# B&R Automation Studio project NAEUL004C00R13L518F00 (part 44)

#### Act_Main.st - Do Not Change!!!
```iecst
(** 2019-10-30 **)
ACTION Act_Main:

	fbInit.bOnDirMod	:= tylocalMagConv2Clp.In.bOnDirMod;
	fbInit.tMtrOffDlyTm	:= tylocalMagConv2Clp.In.tMtrOffDlyTm;
	fbEnt.bOnDirMod		:= tylocalMagConv2Clp.In.bOnDirMod;
	fbEnt.tMtrOffDlyTm	:= tylocalMagConv2Clp.In.tMtrOffDlyTm;
	fbPreExit.bOnDirMod		:= tylocalMagConv2Clp.In.bOnDirMod;
	fbPreExit.tMtrOffDlyTm	:= tylocalMagConv2Clp.In.tMtrOffDlyTm;
	fbExit.bOnDirMod	:= tylocalMagConv2Clp.In.bOnDirMod;
	fbExit.tMtrOffDlyTm	:= tylocalMagConv2Clp.In.tMtrOffDlyTm;
	fbExit1.bOnDirMod		:= tylocalMagConv2Clp.In.bOnDirMod;
	fbExit1.tMtrOffDlyTm	:= tylocalMagConv2Clp.In.tMtrOffDlyTm;
	fbFixClprClampChk.tTimeOut	:= tylocalMagConv2Clp.In.tClprClampTO;
	fbFixClprUnclampChk.tTimeOut	:= tylocalMagConv2Clp.In.tClprUnclampTO;
	fbRmtClprClampChk.tTimeOut	:= tylocalMagConv2Clp.In.tClprClampTO;
	fbRmtClprUnclampChk.tTimeOut	:= tylocalMagConv2Clp.In.tClprUnclampTO;
	fbClprDlyTm.PT	:= tylocalMagConv2Clp.In.tMtrOffDlyTm / 2;
	//Set tylocalMagConv2Clp.In.eAct
	IF tylocalMagConv2Clp.Out.eStatus = Idle OR tylocalMagConv2Clp.Out.eStatus = Busy OR tylocalMagConv2Clp.Out.eStatus = Done THEN
		tylocalMagConv2Clp.Out.eStat	:= tylocalMagConv2Clp.In.eAct;
	END_IF

	IF eStatOld <> tylocalMagConv2Clp.Out.eStat THEN
		fbInit(bEn := FALSE);
		fbEnt(bEn := FALSE);
		fbPreExit(bEn := FALSE);
		fbExit(bEn := FALSE);
		fbExit1(bEn := FALSE);
		fbStop(bEn := FALSE);
		fbFixClprClampChk(bEn := FALSE);
		fbFixClprUnclampChk(bEn := FALSE);
		fbRmtClprClampChk(bEn := FALSE);
		fbRmtClprUnclampChk(bEn := FALSE);
		fbClprDlyTm(IN := FALSE);
		fbFixClprDly(IN := FALSE);
		fbWidthChk(IN := FALSE);
		fbClampTim(IN := FALSE);

		IF eStatOld <> MagConv2ClpActIdle
			AND eStatOld <> MagConv2ClpActSetMtrSigOnOrLToR
			AND eStatOld <> MagConv2ClpActSetMtrDirOrRToL
			AND eStatOld <> MagConv2ClpActRstMtrSigOnOrLToR
			AND eStatOld <> MagConv2ClpActRstMtrDirOrRToL
			AND eStatOld <> MagConv2ClpActSetMtrAll
			AND eStatOld <> MagConv2ClpActRstMtrAll THEN

			tylocalMagConv2Clp.Out.bMtrSigOnOrLToR	:= FALSE;
			tylocalMagConv2Clp.Out.bMtrDirOrRToL	:= FALSE;

		END_IF

		usiStep		:= 0;
		usiSubStep	:= 0;
		usiPrevStep := 0;
		bReachEnd	:= FALSE;

		tylocalMagConv2Clp.Out.sStatTxt	:= a_sStatText[tylocalMagConv2Clp.Out.eStat];

		eStatOld	:= tylocalMagConv2Clp.Out.eStat;

		tylocalMagConv2Clp.Out.eStatus		:= Busy;
	END_IF

	//Main
	CASE tylocalMagConv2Clp.Out.eStat OF

		MagConv2ClpActIdle:
			IF EDGENEG(tylocalMagConv2Clp.In.bManual) THEN
				tylocalMagConv2Clp.Out.bMtrSigOnOrLToR	:= FALSE;
				tylocalMagConv2Clp.Out.bMtrDirOrRToL	:= FALSE;
			END_IF

			tylocalMagConv2Clp.Out.eStatus	:= Idle;

		MagConv2ClpActInit:
			IF tylocalMagConv2Clp.Out.eStatus = Idle OR tylocalMagConv2Clp.Out.eStatus = Busy THEN

				tylocalMagConv2Clp.Out.eStatus	:= Busy;

				//Magazine Conveyor Init Run
				//Detect Have Magazine
				IF tylocalMagConv2Clp.In.bLeftSen OR tylocalMagConv2Clp.In.bRightSen THEN
					tylocalMagConv2Clp.Out.bHvMag	:= TRUE;
				ELSE
					tylocalMagConv2Clp.Out.bHvMag	:= FALSE;
				END_IF

				fbInit.bConvLToR	:= (tylocalMagConv2Clp.In.eDirection = ConvDirLToR) OR (tylocalMagConv2Clp.In.eDirection = ConvDirLToL);
				fbInit.tTxDlyTm		:= DINT_TO_TIME(tylocalMagConv2Clp.In.diInitTm);

				IF fbInit.bConvLToR = TRUE THEN
					fbInit.bEndSen	:= tylocalMagConv2Clp.In.bRightSen;
				ELSE
					fbInit.bEndSen	:= tylocalMagConv2Clp.In.bLeftSen;
				END_IF

				fbInit(bEn := TRUE);

				tylocalMagConv2Clp.Out.bMtrSigOnOrLToR	:= fbInit.bMtrSigOnOrLToR;
				tylocalMagConv2Clp.Out.bMtrDirOrRToL	:= fbInit.bMtrDirOrRToL;

				IF fbInit.udiStatus = 0 THEN
					IF fbInit.bConvLToR = TRUE THEN
						IF tylocalMagConv2Clp.Out.bHvMag = TRUE AND tylocalMagConv2Clp.In.bRightSen = FALSE THEN
							udiStatus	:= 10000;	//Magazine Detected But Not Present At Outlet Sensor (L - R) While Magazine Conveyor Initial
							tylocalMagConv2Clp.Out.eStatus		:= Error;
						ELSE
							tylocalMagConv2Clp.Out.eStatus	:= Done;
						END_IF
					ELSE
						IF tylocalMagConv2Clp.Out.bHvMag = TRUE AND tylocalMagConv2Clp.In.bLeftSen = FALSE THEN
							udiStatus	:= 10001;	//Magazine Detected But Not Present At Outlet Sensor (R - L) While Magazine Conveyor Initial
							tylocalMagConv2Clp.Out.eStatus		:= Error;
						ELSE
							tylocalMagConv2Clp.Out.eStatus	:= Done;
						END_IF
					END_IF
				ELSIF fbInit.udiStatus < 65534 THEN
					udiStatus	:= fbInit.udiStatus;
					tylocalMagConv2Clp.Out.eStatus		:= Error;
				END_IF
			END_IF

		MagConv2ClpActInitStopClp:
			IF tylocalMagConv2Clp.Out.eStatus = Idle OR tylocalMagConv2Clp.Out.eStatus = Busy THEN

				tylocalMagConv2Clp.Out.eStatus	:= Busy;

				CASE usiStep OF
					0:	//Unclamp
						tylocalMagConv2Clp.Out.bFixClprClampCtrl	:= FALSE;
						tylocalMagConv2Clp.Out.bRmtClprClampCtrl	:= FALSE;
						tylocalMagConv2Clp.Out.bFixClprUnClampCtrl	:= TRUE;
						tylocalMagConv2Clp.Out.bRmtClprUnClampCtrl	:= TRUE;

						fbFixClprUnclampChk.bExtSen		:= tylocalMagConv2Clp.In.bFixClprClampSen;
						fbFixClprUnclampChk.bRetSen		:= tylocalMagConv2Clp.In.bFixClprUnclampSen;
						fbFixClprUnclampChk.bRetSafety	:= tylocalMagConv2Clp.In.bFixClprUnclampSafetySen;
						fbFixClprUnclampChk(bEn := TRUE);

						fbRmtClprUnclampChk.bExtSen		:= tylocalMagConv2Clp.In.bRmtClprClampSen;
						fbRmtClprUnclampChk.bRetSen		:= tylocalMagConv2Clp.In.bRmtClprUnclampSen;
						fbRmtClprUnclampChk.bRetSafety	:= tylocalMagConv2Clp.In.bRmtClprUnclampSafetySen;
						fbRmtClprUnclampChk(bEn := TRUE);

						IF fbFixClprUnclampChk.udiStatus = 0 AND fbRmtClprUnclampChk.udiStatus = 0 THEN
							usiStep	:= 1;
						ELSIF (fbFixClprUnclampChk.udiStatus > 0 AND fbFixClprUnclampChk.udiStatus < 65534) OR (fbRmtClprUnclampChk.udiStatus > 0 AND fbRmtClprUnclampChk.udiStatus < 65534) THEN
							tylocalMagConv2Clp.Out.bFixClprClampCtrl	:= FALSE;
							tylocalMagConv2Clp.Out.bRmtClprClampCtrl	:= FALSE;
							tylocalMagConv2Clp.Out.bFixClprUnClampCtrl	:= FALSE;
							tylocalMagConv2Clp.Out.bRmtClprUnClampCtrl	:= FALSE;

							tylocalMagConv2Clp.Out.eStatus	:= Error;

							IF fbFixClprUnclampChk.udiStatus = 1504 OR fbRmtClprUnclampChk.udiStatus = 1504 THEN
								udiStatus	:= 10002;	//Clamper Clamp Sensor Off Time Out In Unclamp Check While Conveyor Initial With Clamper
							ELSIF fbFixClprUnclampChk.udiStatus = 1505 OR fbRmtClprUnclampChk.udiStatus = 1505 THEN
								udiStatus	:= 10003;	//Clamper Unclamp Sensor On Time Out In Unclamp Check While Conveyor Initial With Clamper
							ELSIF fbFixClprUnclampChk.udiStatus = 1508 OR fbRmtClprUnclampChk.udiStatus = 1508 THEN
								udiStatus	:= 10004;	//Clamper Unclamp Safety Sensor Error In Unclamp Check While Conveyor Initial With Clamper
							ELSE
								IF fbFixClprUnclampChk.udiStatus > 0 AND fbFixClprUnclampChk.udiStatus < 65534 THEN
									udiStatus	:= fbFixClprUnclampChk.udiStatus;
								ELSIF fbRmtClprUnclampChk.udiStatus > 0 AND fbRmtClprUnclampChk.udiStatus < 65534 THEN
									udiStatus	:= fbRmtClprUnclampChk.udiStatus;
								END_IF
							END_IF
						END_IF

					1:	//Magazine Conveyor Init Run
						//Detect Have Magazine
						IF tylocalMagConv2Clp.In.bLeftSen OR tylocalMagConv2Clp.In.bRightSen THEN
							tylocalMagConv2Clp.Out.bHvMag	:= TRUE;
						ELSE
							tylocalMagConv2Clp.Out.bHvMag	:= FALSE;
						END_IF

						fbInit.bConvLToR	:= (tylocalMagConv2Clp.In.eDirection = ConvDirLToR) OR (tylocalMagConv2Clp.In.eDirection = ConvDirLToL);
						fbInit.tTxDlyTm		:= DINT_TO_TIME(tylocalMagConv2Clp.In.diInitTm);

						IF fbInit.bConvLToR = TRUE THEN
							fbInit.bEndSen	:= tylocalMagConv2Clp.In.bRightSen;
						ELSE
							fbInit.bEndSen	:= tylocalMagConv2Clp.In.bLeftSen;
						END_IF

						fbInit(bEn := TRUE);

						tylocalMagConv2Clp.Out.bMtrSigOnOrLToR	:= fbInit.bMtrSigOnOrLToR;
						tylocalMagConv2Clp.Out.bMtrDirOrRToL	:= fbInit.bMtrDirOrRToL;

						IF fbInit.udiStatus = 0 THEN
							IF fbInit.bConvLToR = TRUE THEN
								IF tylocalMagConv2Clp.Out.bHvMag = TRUE AND tylocalMagConv2Clp.In.bRightSen = FALSE THEN
									udiStatus	:= 10005;	//Magazine Detected But Not Present At Outlet Sensor (L - R) While Conveyor Initial With Clamper
									tylocalMagConv2Clp.Out.eStatus		:= Error;
								ELSE
									usiStep	:= 2;
								END_IF
							ELSE
								IF tylocalMagConv2Clp.Out.bHvMag = TRUE AND tylocalMagConv2Clp.In.bLeftSen = FALSE THEN
									udiStatus	:= 10006;	//Magazine Detected But Not Present At Outlet Sensor (R - L) While Conveyor Initial With Clamper
									tylocalMagConv2Clp.Out.eStatus		:= Error;
								ELSE
									usiStep	:= 2;
								END_IF
							END_IF
						ELSIF fbInit.udiStatus < 65534 THEN
							udiStatus	:= fbInit.udiStatus;
							tylocalMagConv2Clp.Out.eStatus		:= Error;
						END_IF

					2:	//Check If Have Magazine
						IF tylocalMagConv2Clp.Out.bHvMag = TRUE THEN
							fbWidthChk(IN := NOT tylocalMagConv2Clp.In.bWidthChkInterrupt);
							IF tylocalMagConv2Clp.In.bWidthChkInterrupt = FALSE THEN
								IF fbWidthChk.Q THEN
									udiStatus := 10048;
									tylocalMagConv2Clp.Out.eStatus	  := Error; //Safety Sensor Is Deactivated Before Clamp
								END_IF
							ELSIF tylocalMagConv2Clp.In.bWidthChkInterrupt THEN
								usiStep	  := 3;
							END_IF
						ELSE
							tylocalMagConv2Clp.Out.eStatus	:= Done;
						END_IF

					3:	//Fix Clamp
						tylocalMagConv2Clp.Out.bFixClprClampCtrl	:= TRUE;
						tylocalMagConv2Clp.Out.bFixClprUnClampCtrl	:= FALSE;

						fbFixClprClampChk.bExtSen		:= tylocalMagConv2Clp.In.bFixClprClampSen;
						fbFixClprClampChk.bRetSen		:= tylocalMagConv2Clp.In.bFixClprUnclampSen;
						fbFixClprClampChk.bExtSafety	:= tylocalMagConv2Clp.In.bFixClprClampSafetySen;
						fbFixClprClampChk(bEn := TRUE);

						IF fbFixClprClampChk.udiStatus = 0 THEN
							fbFixClprDly (IN := TRUE);
							IF  fbFixClprDly.Q THEN
								fbFixClprDly (IN := FALSE);
								usiStep	:= 4;
							END_IF

						ELSIF fbFixClprClampChk.udiStatus < 65534 THEN
							tylocalMagConv2Clp.Out.bFixClprClampCtrl	:= FALSE;
							tylocalMagConv2Clp.Out.bFixClprUnClampCtrl	:= FALSE;

							tylocalMagConv2Clp.Out.eStatus	:= Error;

							IF fbFixClprClampChk.udiStatus = 1503 THEN
								udiStatus	:= 10007;	//Clamper Clamp Sensor On Time Out In Clamp Check While Conveyor Initial With Clamper
							ELSIF fbFixClprClampChk.udiStatus = 1506 THEN
								udiStatus	:= 10008;	//Clamper Unclamp Sensor Off Time Out In Clamp Check While Conveyor Initial With Clamper
							ELSIF fbFixClprClampChk.udiStatus = 1507 THEN
								udiStatus	:= 10009;	//Clamper Clamp Safety Sensor Error In Clamp Check While Conveyor Initial With Clamper
							ELSE
								udiStatus	:= fbFixClprClampChk.udiStatus;
							END_IF
						END_IF

					4:	//Remote Clamp
						tylocalMagConv2Clp.Out.bRmtClprClampCtrl	:= TRUE;
						tylocalMagConv2Clp.Out.bRmtClprUnClampCtrl	:= FALSE;

						fbRmtClprClampChk.bExtSen		:= tylocalMagConv2Clp.In.bRmtClprClampSen;
						fbRmtClprClampChk.bRetSen		:= tylocalMagConv2Clp.In.bRmtClprUnclampSen;
						fbRmtClprClampChk.bExtSafety	:= tylocalMagConv2Clp.In.bRmtClprClampSafetySen;
						fbRmtClprClampChk(bEn := TRUE);

						IF fbRmtClprClampChk.udiStatus = 0 THEN
							tylocalMagConv2Clp.Out.eStatus	:= Done;

						ELSIF fbRmtClprClampChk.udiStatus < 65534 THEN
							tylocalMagConv2Clp.Out.bRmtClprClampCtrl	:= FALSE;
							tylocalMagConv2Clp.Out.bRmtClprUnClampCtrl	:= FALSE;
							tylocalMagConv2Clp.Out.eStatus	:= Error;

							IF fbRmtClprClampChk.udiStatus = 1503 THEN
								udiStatus	:= 10007;	//Clamper Clamp Sensor On Time Out In Clamp Check While Conveyor Initial With Clamper
							ELSIF fbRmtClprClampChk.udiStatus = 1506 THEN
								udiStatus	:= 10008;	//Clamper Unclamp Sensor Off Time Out In Clamp Check While Conveyor Initial With Clamper
							ELSIF fbRmtClprClampChk.udiStatus = 1507 THEN
								udiStatus	:= 10009;	//Clamper Clamp Safety Sensor Error In Clamp Check While Conveyor Initial With Clamper
							ELSE
								udiStatus	:= fbRmtClprClampChk.udiStatus;
							END_IF
						END_IF

				END_CASE
			END_IF

		MagConv2ClpActInitClpStop:
			IF tylocalMagConv2Clp.Out.eStatus = Idle OR tylocalMagConv2Clp.Out.eStatus = Busy THEN

				tylocalMagConv2Clp.Out.eStatus	:= Busy;

				CASE usiStep OF
					0:	//Unclamp
						tylocalMagConv2Clp.Out.bFixClprClampCtrl	:= FALSE;
						tylocalMagConv2Clp.Out.bRmtClprClampCtrl	:= FALSE;
						tylocalMagConv2Clp.Out.bFixClprUnClampCtrl	:= TRUE;
						tylocalMagConv2Clp.Out.bRmtClprUnClampCtrl	:= TRUE;

						fbFixClprUnclampChk.bExtSen		:= tylocalMagConv2Clp.In.bFixClprClampSen;
						fbFixClprUnclampChk.bRetSen		:= tylocalMagConv2Clp.In.bFixClprUnclampSen;
						fbFixClprUnclampChk.bRetSafety	:= tylocalMagConv2Clp.In.bFixClprUnclampSafetySen;
						fbFixClprUnclampChk(bEn := TRUE);

						fbRmtClprUnclampChk.bExtSen		:= tylocalMagConv2Clp.In.bRmtClprClampSen;
						fbRmtClprUnclampChk.bRetSen		:= tylocalMagConv2Clp.In.bRmtClprUnclampSen;
						fbRmtClprUnclampChk.bRetSafety	:= tylocalMagConv2Clp.In.bRmtClprUnclampSafetySen;
						fbRmtClprUnclampChk(bEn := TRUE);

						IF fbFixClprUnclampChk.udiStatus = 0 AND fbRmtClprUnclampChk.udiStatus = 0 THEN
							usiStep	:= 1;
						ELSIF (fbFixClprUnclampChk.udiStatus > 0 AND fbFixClprUnclampChk.udiStatus < 65534) OR (fbRmtClprUnclampChk.udiStatus > 0 AND fbRmtClprUnclampChk.udiStatus < 65534) THEN
							tylocalMagConv2Clp.Out.bFixClprClampCtrl	:= FALSE;
							tylocalMagConv2Clp.Out.bRmtClprClampCtrl	:= FALSE;
							tylocalMagConv2Clp.Out.bFixClprUnClampCtrl	:= FALSE;
							tylocalMagConv2Clp.Out.bRmtClprUnClampCtrl	:= FALSE;

							tylocalMagConv2Clp.Out.eStatus	:= Error;

							IF fbFixClprUnclampChk.udiStatus = 1504 OR fbRmtClprUnclampChk.udiStatus = 1504 THEN
								udiStatus	:= 10002;	//Clamper Clamp Sensor Off Time Out In Unclamp Check While Conveyor Initial With Clamper
							ELSIF fbFixClprUnclampChk.udiStatus = 1505 OR fbRmtClprUnclampChk.udiStatus = 1505 THEN
								udiStatus	:= 10003;	//Clamper Unclamp Sensor On Time Out In Unclamp Check While Conveyor Initial With Clamper
							ELSIF fbFixClprUnclampChk.udiStatus = 1508 OR fbRmtClprUnclampChk.udiStatus = 1508 THEN
								udiStatus	:= 10004;	//Clamper Unclamp Safety Sensor Error In Unclamp Check While Conveyor Initial With Clamper
							ELSE
								IF fbFixClprUnclampChk.udiStatus > 0 AND fbFixClprUnclampChk.udiStatus < 65534 THEN
									udiStatus	:= fbFixClprUnclampChk.udiStatus;
								ELSIF fbRmtClprUnclampChk.udiStatus > 0 AND fbRmtClprUnclampChk.udiStatus < 65534 THEN
									udiStatus	:= fbRmtClprUnclampChk.udiStatus;
								END_IF
							END_IF
						END_IF

					1:	//Magazine Conveyor Init Run & Clamp
						//Detect Have Magazine
						IF tylocalMagConv2Clp.In.bLeftSen OR tylocalMagConv2Clp.In.bRightSen THEN
							tylocalMagConv2Clp.Out.bHvMag	:= TRUE;
						ELSE
							tylocalMagConv2Clp.Out.bHvMag	:= FALSE;
						END_IF

						fbInit.bConvLToR	:= (tylocalMagConv2Clp.In.eDirection = ConvDirLToR) OR (tylocalMagConv2Clp.In.eDirection = ConvDirLToL);
						fbInit.tTxDlyTm		:= DINT_TO_TIME(tylocalMagConv2Clp.In.diInitTm);

						IF fbInit.bConvLToR = TRUE THEN
							fbInit.bEndSen	:= tylocalMagConv2Clp.In.bRightSen;
						ELSE
							fbInit.bEndSen	:= tylocalMagConv2Clp.In.bLeftSen;
						END_IF

						fbInit(bEn := TRUE);

						tylocalMagConv2Clp.Out.bMtrSigOnOrLToR	:= fbInit.bMtrSigOnOrLToR;
						tylocalMagConv2Clp.Out.bMtrDirOrRToL	:= fbInit.bMtrDirOrRToL;

						IF fbInit.bEndSen = TRUE THEN
							bReachEnd	:= TRUE;
						END_IF

						IF bReachEnd = TRUE THEN
							fbClprDlyTm(IN := TRUE);
							IF fbClprDlyTm.Q = TRUE THEN
								CASE usiSubStep OF
									//	0:	//Fix Clamp
									//										tylocalMagConv2Clp.Out.bFixClprClampCtrl	:= TRUE;

									//										fbFixClprClampChk.bExtSen		:= tylocalMagConv2Clp.In.bFixClprClampSen;
									//										fbFixClprClampChk.bRetSen		:= tylocalMagConv2Clp.In.bFixClprUnclampSen;
									//										fbFixClprClampChk.bExtSafety	:= tylocalMagConv2Clp.In.bFixClprClampSafetySen;
									//										fbFixClprClampChk(bEn := TRUE);
									//
									//										IF fbFixClprClampChk.udiStatus = 0 THEN
									//											usiSubStep	:= 1;
									//										END_IF

									0:	//Remote Clamp
										tylocalMagConv2Clp.Out.bRmtClprClampCtrl	:= TRUE;
										tylocalMagConv2Clp.Out.bRmtClprUnClampCtrl	:= FALSE;
										fbRmtClprClampChk.bExtSen		:= tylocalMagConv2Clp.In.bRmtClprClampSen;
										fbRmtClprClampChk.bRetSen		:= tylocalMagConv2Clp.In.bRmtClprUnclampSen;
										fbRmtClprClampChk.bExtSafety	:= tylocalMagConv2Clp.In.bRmtClprClampSafetySen;
										fbRmtClprClampChk(bEn := TRUE);

										IF fbRmtClprClampChk.udiStatus = 0 THEN
											usiSubStep	:= 1;
										END_IF

									1:

										tylocalMagConv2Clp.Out.bFixClprClampCtrl	:= TRUE;
										tylocalMagConv2Clp.Out.bFixClprUnClampCtrl	:= FALSE;

										fbFixClprClampChk.bExtSen		:= tylocalMagConv2Clp.In.bFixClprClampSen;
										fbFixClprClampChk.bRetSen		:= tylocalMagConv2Clp.In.bFixClprUnclampSen;
										fbFixClprClampChk.bExtSafety	:= tylocalMagConv2Clp.In.bFixClprClampSafetySen;
										fbFixClprClampChk(bEn := TRUE);

								END_CASE
							END_IF
						END_IF

						IF (fbInit.udiStatus = 0) AND ((fbFixClprClampChk.udiStatus = 0 AND fbRmtClprClampChk.udiStatus = 0) OR (bReachEnd = FALSE)) THEN
							IF fbInit.bConvLToR = TRUE THEN
								IF tylocalMagConv2Clp.Out.bHvMag = TRUE AND tylocalMagConv2Clp.In.bRightSen = FALSE THEN
									udiStatus	:= 10041;	//Magazine Detected But Not Present At Outlet Sensor (L - R) While Conveyor Initial With Clamper
									tylocalMagConv2Clp.Out.eStatus		:= Error;
								ELSE
									tylocalMagConv2Clp.Out.eStatus		:= Done;
								END_IF
							ELSE
								IF tylocalMagConv2Clp.Out.bHvMag = TRUE AND tylocalMagConv2Clp.In.bLeftSen = FALSE THEN
									udiStatus	:= 10042;	//Magazine Detected But Not Present At Outlet Sensor (R - L) While Conveyor Initial With Clamper
									tylocalMagConv2Clp.Out.eStatus		:= Error;
								ELSE
									tylocalMagConv2Clp.Out.eStatus		:= Done;
								END_IF
							END_IF

						ELSIF fbInit.udiStatus > 0 AND fbInit.udiStatus < 65534 THEN
							udiStatus	:= fbInit.udiStatus;
							tylocalMagConv2Clp.Out.eStatus		:= Error;

						ELSIF (fbFixClprClampChk.udiStatus > 0 AND fbFixClprClampChk.udiStatus < 65534) OR (fbRmtClprClampChk.udiStatus > 0 AND fbRmtClprClampChk.udiStatus < 65534) THEN
							tylocalMagConv2Clp.Out.bFixClprClampCtrl	:= FALSE;
							tylocalMagConv2Clp.Out.bRmtClprClampCtrl	:= FALSE;
							tylocalMagConv2Clp.Out.bFixClprUnClampCtrl	:= FALSE;
							tylocalMagConv2Clp.Out.bRmtClprUnClampCtrl	:= FALSE;

							tylocalMagConv2Clp.Out.eStatus	:= Error;

							IF fbFixClprClampChk.udiStatus = 1503 OR fbRmtClprClampChk.udiStatus = 1503 THEN
								udiStatus	:= 10043;	//Clamper Clamp Sensor On Time Out In Clamp Check While Conveyor Initial With Clamper
							ELSIF fbFixClprClampChk.udiStatus = 1506 OR fbRmtClprClampChk.udiStatus = 1506 THEN
								udiStatus	:= 10044;	//Clamper Unclamp Sensor Off Time Out In Clamp Check While Conveyor Initial With Clamper
							ELSIF fbFixClprClampChk.udiStatus = 1507 OR fbRmtClprClampChk.udiStatus = 1507 THEN
								udiStatus	:= 10045;	//Clamper Clamp Safety Sensor Error In Clamp Check While Conveyor Initial With Clamper
							ELSE
								IF fbFixClprClampChk.udiStatus > 0 AND fbFixClprClampChk.udiStatus < 65534 THEN
									udiStatus	:= fbFixClprClampChk.udiStatus;
								ELSIF fbRmtClprClampChk.udiStatus > 0 AND fbRmtClprClampChk.udiStatus < 65534 THEN
									udiStatus	:= fbRmtClprClampChk.udiStatus;
								END_IF
							END_IF
						END_IF

				END_CASE
			END_IF

		MagConv2ClpActEnt:
			IF tylocalMagConv2Clp.Out.eStatus = Idle OR tylocalMagConv2Clp.Out.eStatus = Busy THEN

				tylocalMagConv2Clp.Out.eStatus	:= Busy;

				//Detect Have Magazine
				IF tylocalMagConv2Clp.In.bLeftSen OR tylocalMagConv2Clp.In.bRightSen THEN
					tylocalMagConv2Clp.Out.bHvMag	:= TRUE;
				END_IF

				//Conveyor Run
				fbEnt.bConvLToR		:= (tylocalMagConv2Clp.In.eDirection = ConvDirLToR) OR (tylocalMagConv2Clp.In.eDirection = ConvDirLToL);
				fbEnt.tTimeOut		:= DINT_TO_TIME(tylocalMagConv2Clp.In.diTxInTimeOut);

				IF fbEnt.bConvLToR = TRUE THEN
					fbEnt.bEndSen	:= tylocalMagConv2Clp.In.bRightSen;
				ELSE
					fbEnt.bEndSen	:= tylocalMagConv2Clp.In.bLeftSen;
				END_IF

				fbEnt(bEn := TRUE);

				tylocalMagConv2Clp.Out.bMtrSigOnOrLToR	:= fbEnt.bMtrSigOnOrLToR;
				tylocalMagConv2Clp.Out.bMtrDirOrRToL	:= fbEnt.bMtrDirOrRToL;

				IF fbEnt.udiStatus = 0 THEN
					tylocalMagConv2Clp.Out.eStatus		:= Done;
				ELSIF fbEnt.udiStatus < 65534 THEN
					tylocalMagConv2Clp.Out.eStatus		:= Error;

					IF fbEnt.udiStatus = 1101 THEN
						udiStatus	:= 10028;	//Transfer In Time Out While Entering Magazine
					ELSE
						udiStatus	:= fbEnt.udiStatus;
					END_IF
				END_IF

			END_IF

		MagConv2ClpActEntStopClp:
			IF tylocalMagConv2Clp.Out.eStatus = Idle OR tylocalMagConv2Clp.Out.eStatus = Busy THEN

				tylocalMagConv2Clp.Out.eStatus	:= Busy;

				CASE usiStep OF
					0:	//Conveyor Enter
						//Detect Have Magazine
						IF tylocalMagConv2Clp.In.bLeftSen OR tylocalMagConv2Clp.In.bRightSen THEN
							tylocalMagConv2Clp.Out.bHvMag	:= TRUE;
						END_IF

						//Conveyor Run
						fbEnt.bConvLToR		:= (tylocalMagConv2Clp.In.eDirection = ConvDirLToR) OR (tylocalMagConv2Clp.In.eDirection = ConvDirLToL);
						fbEnt.tTimeOut		:= DINT_TO_TIME(tylocalMagConv2Clp.In.diTxInTimeOut);

						IF fbEnt.bConvLToR = TRUE THEN
							fbEnt.bEndSen	:= tylocalMagConv2Clp.In.bRightSen;
						ELSE
							fbEnt.bEndSen	:= tylocalMagConv2Clp.In.bLeftSen;
						END_IF

						fbEnt(bEn := TRUE);

						tylocalMagConv2Clp.Out.bMtrSigOnOrLToR	:= fbEnt.bMtrSigOnOrLToR;
						tylocalMagConv2Clp.Out.bMtrDirOrRToL	:= fbEnt.bMtrDirOrRToL;

						IF fbEnt.udiStatus = 0 THEN
							usiStep	:= 2;
							tRemainingTime := tylocalMagConv2Clp.In.tClprClampTO;

						ELSIF fbEnt.udiStatus < 65534 THEN
							tylocalMagConv2Clp.Out.eStatus	:= Error;

							IF fbEnt.udiStatus = 1101 THEN
								udiStatus	:= 10029;	//Transfer In Time Out While Entering Magazine
							ELSE
								udiStatus	:= fbEnt.udiStatus;
							END_IF
						END_IF
					1: //clamp standby step
						fbFixClprClampChk(bEn:= FALSE);
						fbRmtClprClampChk(bEn:= FALSE);
						fbFixClprUnclampChk(bEn:= FALSE);
						fbRmtClprUnclampChk(bEn := FALSE);
						fbInterrupSenDlyOff(IN:= tylocalMagConv2Clp.In.bWidthChkInterrupt);
						IF fbInterrupSenDlyOff.Q THEN
							IF NOT(tylocalMagConv2Clp.In.bLeftSen) AND NOT(tylocalMagConv2Clp.In.bRightSen) THEN
								tylocalMagConv2Clp.Out.eStatus := Error;
								udiStatus	:= 10049; //Magazine is taken away during the clamp
							ELSIF (tylocalMagConv2Clp.In.bLeftSen AND NOT(tylocalMagConv2Clp.In.bRightSen)) THEN
								fbEnt(bEn := FALSE);
								usiStep := 4;
								IF usiPrevStep <> usiStep THEN
									tRemainingTime := tylocalMagConv2Clp.In.tClprClampTO;
								END_IF
							ELSE
								usiStep := usiPrevStep;
								usiPrevStep := 1;
							END_IF
						END_IF

					2:	//Fix Clamp
						tylocalMagConv2Clp.Out.bFixClprClampCtrl	:= TRUE;
						tylocalMagConv2Clp.Out.bFixClprUnClampCtrl	:= FALSE;

						fbFixClprClampChk.bExtSen		:= tylocalMagConv2Clp.In.bFixClprClampSen;
						fbFixClprClampChk.bRetSen		:= tylocalMagConv2Clp.In.bFixClprUnclampSen ;// OR (usiPrevStep = 1 AND tylocalMagConv2Clp.In.bFixClprClampSen = FALSE);
						fbFixClprClampChk.bExtSafety	:= tylocalMagConv2Clp.In.bFixClprClampSafetySen;
						fbFixClprClampChk(bEn := TRUE);
						IF (tRemainingTime) > T#5s THEN
							fbClampTim(IN:= TRUE,PT:= tRemainingTime );
						ELSE
							fbClampTim(IN:= TRUE,PT:= T#6s);
						END_IF
						IF fbFixClprClampChk.udiStatus = 0 THEN
							fbFixClprDly(IN := TRUE);
							IF  fbFixClprDly.Q THEN
								fbFixClprDly (IN := FALSE);
								usiStep	:= 3;
								tRemainingTime := tylocalMagConv2Clp.In.tClprClampTO;
								fbClampTim(IN:= FALSE);
							END_IF
						ELSIF fbFixClprClampChk.udiStatus < 65534 OR fbClampTim.Q THEN
							tylocalMagConv2Clp.Out.bFixClprClampCtrl	:= FALSE;
							tylocalMagConv2Clp.Out.bFixClprUnClampCtrl := FALSE;

							tylocalMagConv2Clp.Out.eStatus	:= Error;

							IF fbFixClprClampChk.udiStatus = 1503 THEN
								udiStatus	:= 10010;	//Clamper Clamp Sensor On Time Out In Clamp Check While Conveyor Enter With Clamper
							ELSIF fbFixClprClampChk.udiStatus = 1506 THEN
								udiStatus	:= 10011;	//Clamper Unclamp Sensor Off Time Out In Clamp Check While Conveyor Enter With Clamper
							ELSIF fbFixClprClampChk.udiStatus = 1507 THEN
								udiStatus	:= 10012;	//Clamper Clamp Safety Sensor Error In Clamp Check While Conveyor Enter With Clamper
							ELSIF fbFixClprClampChk.udiStatus = 65535 AND fbClampTim.Q THEN
								udiStatus	:= 10050;	//Clamper Clamp Sensor On Time Out While Continue to Clamp
							ELSE
								udiStatus	:= fbFixClprClampChk.udiStatus;
							END_IF
						ELSIF NOT(tylocalMagConv2Clp.In.bWidthChkInterrupt) THEN
							tylocalMagConv2Clp.Out.bFixClprClampCtrl	:= FALSE;
							tylocalMagConv2Clp.Out.bFixClprUnClampCtrl := FALSE;
							usiPrevStep := 2;
							usiStep	:= 1;
							tRemainingTime := tRemainingTime - fbClampTim.ET;
							fbClampTim(IN:= FALSE);
						END_IF

					3:	//Remote Clamp
						tylocalMagConv2Clp.Out.bRmtClprClampCtrl	:= TRUE;
						tylocalMagConv2Clp.Out.bRmtClprUnClampCtrl	:= FALSE;
						fbRmtClprClampChk.bExtSen		:= tylocalMagConv2Clp.In.bRmtClprClampSen;
						fbRmtClprClampChk.bRetSen		:= tylocalMagConv2Clp.In.bRmtClprUnclampSen ;
						fbRmtClprClampChk.bExtSafety	:= tylocalMagConv2Clp.In.bRmtClprClampSafetySen;
						fbRmtClprClampChk(bEn := TRUE);
						IF (tRemainingTime ) > T#6s THEN
							fbClampTim(IN:= TRUE,PT:= tRemainingTime );
						ELSE
							fbClampTim(IN:= TRUE,PT:= T#5s);
						END_IF
						IF fbRmtClprClampChk.udiStatus = 0 THEN
							tylocalMagConv2Clp.Out.eStatus	:= Done;
						ELSIF fbRmtClprClampChk.udiStatus < 65534 OR fbClampTim.Q THEN
							tylocalMagConv2Clp.Out.bRmtClprClampCtrl	:= FALSE;
							tylocalMagConv2Clp.Out.bRmtClprUnClampCtrl	:= FALSE;
							tylocalMagConv2Clp.Out.eStatus	:= Error;

							IF fbRmtClprClampChk.udiStatus = 1503 THEN
								udiStatus	:= 10010;	//Clamper Clamp Sensor On Time Out In Clamp Check While Conveyor Enter With Clamper
							ELSIF fbRmtClprClampChk.udiStatus = 1506 THEN
								udiStatus	:= 10011;	//Clamper Unclamp Sensor Off Time Out In Clamp Check While Conveyor Enter With Clamper
							ELSIF fbRmtClprClampChk.udiStatus = 1507 THEN
								udiStatus	:= 10012;	//Clamper Clamp Safety Sensor Error In Clamp Check While Conveyor Enter With Clamper
							ELSIF fbRmtClprClampChk.udiStatus = 65535 AND fbClampTim.Q THEN
								udiStatus	:= 10051;	//Clamper Clamp Sensor On Time Out While Continue to Clamp
							ELSE
								udiStatus	:= fbRmtClprClampChk.udiStatus;
							END_IF
						ELSIF NOT(tylocalMagConv2Clp.In.bWidthChkInterrupt) THEN
							tylocalMagConv2Clp.Out.bRmtClprClampCtrl	:= FALSE;
							tylocalMagConv2Clp.Out.bRmtClprUnClampCtrl := FALSE;
							usiPrevStep := 3;
							usiStep	:= 1;
							tRemainingTime := tRemainingTime - fbClampTim.ET;
							fbClampTim(IN:= FALSE);
						END_IF
					4:
						tylocalMagConv2Clp.Out.bFixClprClampCtrl	:= FALSE;
						tylocalMagConv2Clp.Out.bRmtClprClampCtrl	:= FALSE;
						tylocalMagConv2Clp.Out.bFixClprUnClampCtrl	:= TRUE;
						tylocalMagConv2Clp.Out.bRmtClprUnClampCtrl	:= TRUE;

						fbFixClprUnclampChk.bExtSen		:= tylocalMagConv2Clp.In.bFixClprClampSen;
						fbFixClprUnclampChk.bRetSen		:= tylocalMagConv2Clp.In.bFixClprUnclampSen;
						fbFixClprUnclampChk.bRetSafety	:= tylocalMagConv2Clp.In.bFixClprUnclampSafetySen;
						fbFixClprUnclampChk(bEn := TRUE);

						fbRmtClprUnclampChk.bExtSen		:= tylocalMagConv2Clp.In.bRmtClprClampSen;
						fbRmtClprUnclampChk.bRetSen		:= tylocalMagConv2Clp.In.bRmtClprUnclampSen;
						fbRmtClprUnclampChk.bRetSafety	:= tylocalMagConv2Clp.In.bRmtClprUnclampSafetySen;
						fbRmtClprUnclampChk(bEn := TRUE);
						IF (tRemainingTime) > T#5s THEN
							fbClampTim(IN:= TRUE,PT:= tRemainingTime );
						ELSE
							fbClampTim(IN:= TRUE,PT:= T#6s);
						END_IF
						IF fbFixClprUnclampChk.udiStatus = 0 AND fbRmtClprUnclampChk.udiStatus = 0 THEN
							usiStep := 0;
							tRemainingTime := tylocalMagConv2Clp.In.tClprClampTO;
							fbClampTim(IN:= FALSE);
						ELSIF (fbFixClprUnclampChk.udiStatus > 0 AND fbFixClprUnclampChk.udiStatus < 65534) OR (fbRmtClprUnclampChk.udiStatus > 0 AND fbRmtClprUnclampChk.udiStatus < 65534) OR fbClampTim.Q THEN
							tylocalMagConv2Clp.Out.bFixClprClampCtrl	:= FALSE;
							tylocalMagConv2Clp.Out.bRmtClprClampCtrl	:= FALSE;
							tylocalMagConv2Clp.Out.bFixClprUnClampCtrl	:= FALSE;
							tylocalMagConv2Clp.Out.bRmtClprUnClampCtrl	:= FALSE;

							tylocalMagConv2Clp.Out.eStatus	:= Error;

							IF fbFixClprUnclampChk.udiStatus = 1504 OR fbRmtClprUnclampChk.udiStatus = 1504 THEN
								udiStatus	:= 10002;	//Clamper Clamp Sensor Off Time Out In Unclamp Check While Conveyor Initial With Clamper
							ELSIF fbFixClprUnclampChk.udiStatus = 1505 OR fbRmtClprUnclampChk.udiStatus = 1505 THEN
								udiStatus	:= 10003;	//Clamper Unclamp Sensor On Time Out In Unclamp Check While Conveyor Initial With Clamper
							ELSIF fbFixClprUnclampChk.udiStatus = 1508 OR fbRmtClprUnclampChk.udiStatus = 1508 THEN
								udiStatus	:= 10004;	//Clamper Unclamp Safety Sensor Error In Unclamp Check While Conveyor Initial With Clamper
							ELSIF fbFixClprUnclampChk.udiStatus > 0 AND fbFixClprUnclampChk.udiStatus < 65534 THEN
								udiStatus	:= fbFixClprUnclampChk.udiStatus;
							ELSIF fbRmtClprUnclampChk.udiStatus > 0 AND fbRmtClprUnclampChk.udiStatus < 65534 THEN
								udiStatus	:= fbRmtClprUnclampChk.udiStatus;
							ELSIF (fbFixClprUnclampChk.udiStatus = 65535 AND fbRmtClprUnclampChk.udiStatus = 65535) OR fbClampTim.Q THEN
								udiStatus	:= 10052;	//Clamper Unclamp Sensor On Time Out While Continue to UnClamp
							END_IF
						ELSIF NOT(tylocalMagConv2Clp.In.bWidthChkInterrupt) THEN
							tylocalMagConv2Clp.Out.bRmtClprClampCtrl	:= FALSE;
							tylocalMagConv2Clp.Out.bRmtClprUnClampCtrl := FALSE;
							usiPrevStep := 4;
							usiStep	:= 1;
							tRemainingTime := tRemainingTime - fbClampTim.ET;
							fbClampTim(IN:= FALSE);
						END_IF
				END_CASE

			END_IF

		MagConv2ClpActEntClpStop:
			IF tylocalMagConv2Clp.Out.eStatus = Idle OR tylocalMagConv2Clp.Out.eStatus = Busy THEN

				tylocalMagConv2Clp.Out.eStatus	:= Busy;

				//Detect Have Magazine
				IF tylocalMagConv2Clp.In.bLeftSen OR tylocalMagConv2Clp.In.bRightSen THEN
					tylocalMagConv2Clp.Out.bHvMag	:= TRUE;
				END_IF

				//Conveyor Run
				fbEnt.bConvLToR		:= (tylocalMagConv2Clp.In.eDirection = ConvDirLToR) OR (tylocalMagConv2Clp.In.eDirection = ConvDirLToL);
				fbEnt.tTimeOut		:= DINT_TO_TIME(tylocalMagConv2Clp.In.diTxInTimeOut);

				IF fbEnt.bConvLToR = TRUE THEN
					fbEnt.bEndSen	:= tylocalMagConv2Clp.In.bRightSen;
				ELSE
					fbEnt.bEndSen	:= tylocalMagConv2Clp.In.bLeftSen;
				END_IF

				fbEnt(bEn := TRUE);

				tylocalMagConv2Clp.Out.bMtrSigOnOrLToR	:= fbEnt.bMtrSigOnOrLToR;
				tylocalMagConv2Clp.Out.bMtrDirOrRToL	:= fbEnt.bMtrDirOrRToL;

				IF fbEnt.bEndSen = TRUE THEN
					bReachEnd	:= TRUE;
				END_IF

				IF bReachEnd = TRUE THEN
					fbClprDlyTm(IN := TRUE);
					IF fbClprDlyTm.Q = TRUE THEN
						CASE usiSubStep OF
							0:	//Fix Clamp
								//								tylocalMagConv2Clp.Out.bFixClprClampCtrl	:= TRUE;
								//
								//								fbFixClprClampChk.bExtSen		:= tylocalMagConv2Clp.In.bFixClprClampSen;
								//								fbFixClprClampChk.bRetSen		:= tylocalMagConv2Clp.In.bFixClprUnclampSen;
								//								fbFixClprClampChk.bExtSafety	:= tylocalMagConv2Clp.In.bFixClprClampSafetySen;
								//								fbFixClprClampChk(bEn := TRUE);
								//
								//								IF fbFixClprClampChk.udiStatus = 0 THEN
								//									usiSubStep	:= 1;
								//								END_IF

								tylocalMagConv2Clp.Out.bRmtClprClampCtrl	:= TRUE;
								tylocalMagConv2Clp.Out.bRmtClprUnClampCtrl	:= FALSE;
								fbRmtClprClampChk.bExtSen		:= tylocalMagConv2Clp.In.bRmtClprClampSen;
								fbRmtClprClampChk.bRetSen		:= tylocalMagConv2Clp.In.bRmtClprUnclampSen;
								fbRmtClprClampChk.bExtSafety	:= tylocalMagConv2Clp.In.bRmtClprClampSafetySen;
								fbRmtClprClampChk(bEn := TRUE);

								IF fbRmtClprClampChk.udiStatus = 0 THEN
									usiSubStep	:= 1;
								END_IF

							1:	//Remote Clamp
								//								tylocalMagConv2Clp.Out.bRmtClprClampCtrl	:= TRUE;
								//
								//								fbRmtClprClampChk.bExtSen		:= tylocalMagConv2Clp.In.bRmtClprClampSen;
								//								fbRmtClprClampChk.bRetSen		:= tylocalMagConv2Clp.In.bRmtClprUnclampSen;
								//								fbRmtClprClampChk.bExtSafety	:= tylocalMagConv2Clp.In.bRmtClprClampSafetySen;
								//								fbRmtClprClampChk(bEn := TRUE);

								tylocalMagConv2Clp.Out.bFixClprClampCtrl	:= TRUE;
								tylocalMagConv2Clp.Out.bFixClprUnClampCtrl := FALSE;

								fbFixClprClampChk.bExtSen		:= tylocalMagConv2Clp.In.bFixClprClampSen;
								fbFixClprClampChk.bRetSen		:= tylocalMagConv2Clp.In.bFixClprUnclampSen;
								fbFixClprClampChk.bExtSafety	:= tylocalMagConv2Clp.In.bFixClprClampSafetySen;
								fbFixClprClampChk(bEn := TRUE);

						END_CASE
					END_IF
				END_IF

				IF fbEnt.udiStatus = 0 AND (fbFixClprClampChk.udiStatus = 0 AND fbRmtClprClampChk.udiStatus = 0) THEN
					tylocalMagConv2Clp.Out.eStatus	:= Done;

				ELSIF (fbFixClprClampChk.udiStatus > 0 AND fbFixClprClampChk.udiStatus < 65534) OR (fbRmtClprClampChk.udiStatus > 0 AND fbRmtClprClampChk.udiStatus < 65534) THEN
					tylocalMagConv2Clp.Out.bFixClprClampCtrl	:= FALSE;
					tylocalMagConv2Clp.Out.bRmtClprClampCtrl	:= FALSE;
					tylocalMagConv2Clp.Out.bFixClprUnClampCtrl	:= FALSE;
					tylocalMagConv2Clp.Out.bRmtClprUnClampCtrl	:= FALSE;

					tylocalMagConv2Clp.Out.eStatus	:= Error;

					IF fbFixClprClampChk.udiStatus = 1503 OR fbRmtClprClampChk.udiStatus = 1503 THEN
						udiStatus	:= 10034;	//Clamper Clamp Sensor On Time Out In Clamp Check While Conveyor Enter With Clamper
					ELSIF fbFixClprClampChk.udiStatus = 1506 OR fbRmtClprClampChk.udiStatus = 1506 THEN
						udiStatus	:= 10035;	//Clamper Unclamp Sensor Off Time Out In Clamp Check While Conveyor Enter With Clamper
					ELSIF fbFixClprClampChk.udiStatus = 1507 OR fbRmtClprClampChk.udiStatus = 1507 THEN
						udiStatus	:= 10036;	//Clamper Clamp Safety Sensor Error In Clamp Check While Conveyor Enter With Clamper
					ELSE
						IF fbFixClprClampChk.udiStatus > 0 AND fbFixClprClampChk.udiStatus < 65534 THEN
							udiStatus	:= fbFixClprClampChk.udiStatus;
						ELSIF fbRmtClprClampChk.udiStatus > 0 AND fbRmtClprClampChk.udiStatus < 65534 THEN
							udiStatus	:= fbRmtClprClampChk.udiStatus;
						END_IF
					END_IF

				ELSIF fbEnt.udiStatus > 0 AND fbEnt.udiStatus < 65534 THEN
					tylocalMagConv2Clp.Out.eStatus	:= Error;

					IF fbEnt.udiStatus = 1101 THEN
						udiStatus	:= 10037;	//Transfer In Time Out While Entering Magazine
					ELSE
						udiStatus	:= fbEnt.udiStatus;
					END_IF

				END_IF

			END_IF

		MagConv2ClpActPreExit:
			IF tylocalMagConv2Clp.Out.eStatus = Idle OR tylocalMagConv2Clp.Out.eStatus = Busy THEN

				tylocalMagConv2Clp.Out.eStatus	:= Busy;

				//Conveyor Run
				fbPreExit.bConvLToR		:= (tylocalMagConv2Clp.In.eDirection = ConvDirLToR) OR (tylocalMagConv2Clp.In.eDirection = ConvDirRToR);
				fbPreExit.tTxDlyTm		:= DINT_TO_TIME(tylocalMagConv2Clp.In.diInitTm);

				IF fbPreExit.bConvLToR = TRUE THEN
					fbPreExit.bEndSen	:= tylocalMagConv2Clp.In.bRightSen;
					fbPreExit.bStartSen	:= tylocalMagConv2Clp.In.bLeftSen;
				ELSE
					fbPreExit.bEndSen	:= tylocalMagConv2Clp.In.bLeftSen;
					fbPreExit.bStartSen	:= tylocalMagConv2Clp.In.bRightSen;
				END_IF

				fbPreExit(bEn := TRUE);

				tylocalMagConv2Clp.Out.bMtrSigOnOrLToR	:= fbPreExit.bMtrSigOnOrLToR;
				tylocalMagConv2Clp.Out.bMtrDirOrRToL	:= fbPreExit.bMtrDirOrRToL;

				IF fbPreExit.udiStatus = 0 THEN
					IF fbPreExit.bEndSen = TRUE THEN
						tylocalMagConv2Clp.Out.eStatus	:= Done;
					ELSE
						udiStatus	:= 10046;	//Magazine Not Detected While Pre-Exiting Magazine
						tylocalMagConv2Clp.Out.eStatus		:= Error;
					END_IF
				ELSIF fbPreExit.udiStatus < 65534 THEN
					udiStatus	:= fbPreExit.udiStatus;
					tylocalMagConv2Clp.Out.eStatus		:= Error;
				END_IF

			END_IF

		MagConv2ClpActPreExitClpr:
			IF tylocalMagConv2Clp.Out.eStatus = Idle OR tylocalMagConv2Clp.Out.eStatus = Busy THEN

				tylocalMagConv2Clp.Out.eStatus	:= Busy;

				CASE usiStep OF
					0:	//Unclamp
						tylocalMagConv2Clp.Out.bFixClprClampCtrl	:= FALSE;
						tylocalMagConv2Clp.Out.bRmtClprClampCtrl	:= FALSE;
						tylocalMagConv2Clp.Out.bFixClprUnClampCtrl	:= TRUE;
						tylocalMagConv2Clp.Out.bRmtClprUnClampCtrl	:= TRUE;

						fbFixClprUnclampChk.bExtSen		:= tylocalMagConv2Clp.In.bFixClprClampSen;
						fbFixClprUnclampChk.bRetSen		:= tylocalMagConv2Clp.In.bFixClprUnclampSen;
						fbFixClprUnclampChk.bRetSafety	:= tylocalMagConv2Clp.In.bFixClprUnclampSafetySen;
						fbFixClprUnclampChk(bEn := TRUE);

						fbRmtClprUnclampChk.bExtSen		:= tylocalMagConv2Clp.In.bRmtClprClampSen;
						fbRmtClprUnclampChk.bRetSen		:= tylocalMagConv2Clp.In.bRmtClprUnclampSen;
						fbRmtClprUnclampChk.bRetSafety	:= tylocalMagConv2Clp.In.bRmtClprUnclampSafetySen;
						fbRmtClprUnclampChk(bEn := TRUE);

						IF fbFixClprUnclampChk.udiStatus = 0 AND fbRmtClprUnclampChk.udiStatus = 0 THEN
							usiStep	:= 1;
						ELSIF (fbFixClprUnclampChk.udiStatus > 0 AND fbFixClprUnclampChk.udiStatus < 65534) OR (fbRmtClprUnclampChk.udiStatus > 0 AND fbRmtClprUnclampChk.udiStatus < 65534) THEN
							tylocalMagConv2Clp.Out.bFixClprClampCtrl	:= FALSE;
							tylocalMagConv2Clp.Out.bRmtClprClampCtrl	:= FALSE;
							tylocalMagConv2Clp.Out.bFixClprUnClampCtrl	:= FALSE;
							tylocalMagConv2Clp.Out.bRmtClprUnClampCtrl	:= FALSE;

							tylocalMagConv2Clp.Out.eStatus	:= Error;

							IF fbFixClprUnclampChk.udiStatus = 1504 OR fbRmtClprUnclampChk.udiStatus = 1504 THEN
								udiStatus	:= 10002;	//Clamper Clamp Sensor Off Time Out In Unclamp Check While Conveyor Initial With Clamper
							ELSIF fbFixClprUnclampChk.udiStatus = 1505 OR fbRmtClprUnclampChk.udiStatus = 1505 THEN
								udiStatus	:= 10003;	//Clamper Unclamp Sensor On Time Out In Unclamp Check While Conveyor Initial With Clamper
							ELSIF fbFixClprUnclampChk.udiStatus = 1508 OR fbRmtClprUnclampChk.udiStatus = 1508 THEN
								udiStatus	:= 10004;	//Clamper Unclamp Safety Sensor Error In Unclamp Check While Conveyor Initial With Clamper
							ELSE
								IF fbFixClprUnclampChk.udiStatus > 0 AND fbFixClprUnclampChk.udiStatus < 65534 THEN
									udiStatus	:= fbFixClprUnclampChk.udiStatus;
								ELSIF fbRmtClprUnclampChk.udiStatus > 0 AND fbRmtClprUnclampChk.udiStatus < 65534 THEN
									udiStatus	:= fbRmtClprUnclampChk.udiStatus;
								END_IF
							END_IF
						END_IF

					1:	//Conveyor Pre-Exit
						//Conveyor Run
						fbPreExit.bConvLToR		:= (tylocalMagConv2Clp.In.eDirection = ConvDirLToR) OR (tylocalMagConv2Clp.In.eDirection = ConvDirRToR);
						fbPreExit.tTxDlyTm		:= DINT_TO_TIME(tylocalMagConv2Clp.In.diInitTm);

						IF fbPreExit.bConvLToR = TRUE THEN
							fbPreExit.bEndSen	:= tylocalMagConv2Clp.In.bRightSen;
							fbPreExit.bStartSen	:= tylocalMagConv2Clp.In.bLeftSen;
						ELSE
							fbPreExit.bEndSen	:= tylocalMagConv2Clp.In.bLeftSen;
							fbPreExit.bStartSen	:= tylocalMagConv2Clp.In.bRightSen;
						END_IF

						fbPreExit(bEn := TRUE);

						tylocalMagConv2Clp.Out.bMtrSigOnOrLToR	:= fbPreExit.bMtrSigOnOrLToR;
						tylocalMagConv2Clp.Out.bMtrDirOrRToL	:= fbPreExit.bMtrDirOrRToL;

						IF fbPreExit.udiStatus = 0 THEN
							IF fbPreExit.bEndSen = TRUE THEN
								tylocalMagConv2Clp.Out.eStatus	:= Done;
							ELSE
								udiStatus	:= 10046;	//Magazine Not Detected While Pre-Exiting Magazine
								tylocalMagConv2Clp.Out.eStatus		:= Error;
							END_IF
						ELSIF fbPreExit.udiStatus < 65534 THEN
							udiStatus	:= fbPreExit.udiStatus;
							tylocalMagConv2Clp.Out.eStatus		:= Error;
						END_IF

				END_CASE

			END_IF

		MagConv2ClpActExit:
			IF tylocalMagConv2Clp.Out.eStatus = Idle OR tylocalMagConv2Clp.Out.eStatus = Busy THEN

				tylocalMagConv2Clp.Out.eStatus	:= Busy;

				//Conveyor Run
				fbExit.bConvLToR	:= (tylocalMagConv2Clp.In.eDirection = ConvDirLToR) OR (tylocalMagConv2Clp.In.eDirection = ConvDirRToR);
				fbExit.tTimeOut		:= DINT_TO_TIME(tylocalMagConv2Clp.In.diTxOutTimeOut);

				IF fbExit.bConvLToR = TRUE THEN
					fbExit.bEndSen	:= tylocalMagConv2Clp.In.bRightSen;
				ELSE
					fbExit.bEndSen	:= tylocalMagConv2Clp.In.bLeftSen;
				END_IF

				fbExit(bEn := TRUE);

				tylocalMagConv2Clp.Out.bMtrSigOnOrLToR	:= fbExit.bMtrSigOnOrLToR;
				tylocalMagConv2Clp.Out.bMtrDirOrRToL	:= fbExit.bMtrDirOrRToL;

				IF fbExit.udiStatus = 0 THEN
					tylocalMagConv2Clp.Out.bHvMag		:= FALSE;
					tylocalMagConv2Clp.Out.eStatus		:= Done;
				ELSIF fbExit.udiStatus < 65534 THEN
					tylocalMagConv2Clp.Out.eStatus		:= Error;

					IF fbExit.udiStatus = 1101 THEN
						udiStatus	:= 10030;	//Transfer Out Time Out While Exiting Magazine
					ELSE
						udiStatus	:= fbExit.udiStatus;
					END_IF
				END_IF

			END_IF

		MagConv2ClpActExit1:
			IF tylocalMagConv2Clp.Out.eStatus = Idle OR tylocalMagConv2Clp.Out.eStatus = Busy THEN

				tylocalMagConv2Clp.Out.eStatus	:= Busy;

				//Conveyor Run
				fbExit1.bConvLToR		:= (tylocalMagConv2Clp.In.eDirection = ConvDirLToR) OR (tylocalMagConv2Clp.In.eDirection = ConvDirRToR);
				fbExit1.tTimeOut		:= DINT_TO_TIME(tylocalMagConv2Clp.In.diTxOutTimeOut);

				IF fbExit1.bConvLToR = TRUE THEN
					fbExit1.bEndSen	:= tylocalMagConv2Clp.In.bRightSen;
				ELSE
					fbExit1.bEndSen	:= tylocalMagConv2Clp.In.bLeftSen;
				END_IF

				fbExit1(bEn := TRUE);

				tylocalMagConv2Clp.Out.bMtrSigOnOrLToR	:= fbExit1.bMtrSigOnOrLToR;
				tylocalMagConv2Clp.Out.bMtrDirOrRToL	:= fbExit1.bMtrDirOrRToL;

				IF fbExit1.udiStatus = 0 THEN
					tylocalMagConv2Clp.Out.bHvMag		:= FALSE;
					tylocalMagConv2Clp.Out.eStatus		:= Done;
				ELSIF fbExit1.udiStatus < 65534 THEN
					tylocalMagConv2Clp.Out.eStatus		:= Error;

					IF fbExit1.udiStatus = 1101 THEN
						udiStatus	:= 10032;	//Transfer Out Time Out While Exiting Magazinie
					ELSE
						udiStatus	:= fbExit1.udiStatus;
					END_IF
				END_IF

			END_IF

		MagConv2ClpActExitClpr:
			IF tylocalMagConv2Clp.Out.eStatus = Idle OR tylocalMagConv2Clp.Out.eStatus = Busy THEN

				tylocalMagConv2Clp.Out.eStatus	:= Busy;

				CASE usiStep OF
					0:	//Unclamp
						tylocalMagConv2Clp.Out.bFixClprClampCtrl	:= FALSE;
						tylocalMagConv2Clp.Out.bRmtClprClampCtrl	:= FALSE;
						tylocalMagConv2Clp.Out.bFixClprUnClampCtrl	:= TRUE;
						tylocalMagConv2Clp.Out.bRmtClprUnClampCtrl	:= TRUE;

						fbFixClprUnclampChk.bExtSen		:= tylocalMagConv2Clp.In.bFixClprClampSen;
						fbFixClprUnclampChk.bRetSen		:= tylocalMagConv2Clp.In.bFixClprUnclampSen;
						fbFixClprUnclampChk.bRetSafety	:= tylocalMagConv2Clp.In.bFixClprUnclampSafetySen;
						fbFixClprUnclampChk(bEn := TRUE);

						fbRmtClprUnclampChk.bExtSen		:= tylocalMagConv2Clp.In.bRmtClprClampSen;
						fbRmtClprUnclampChk.bRetSen		:= tylocalMagConv2Clp.In.bRmtClprUnclampSen;
						fbRmtClprUnclampChk.bRetSafety	:= tylocalMagConv2Clp.In.bRmtClprUnclampSafetySen;
						fbRmtClprUnclampChk(bEn := TRUE);

						IF fbFixClprUnclampChk.udiStatus = 0 AND fbRmtClprUnclampChk.udiStatus = 0 THEN
							usiStep	:= 1;
						ELSIF (fbFixClprUnclampChk.udiStatus > 0 AND fbFixClprUnclampChk.udiStatus < 65534) OR (fbRmtClprUnclampChk.udiStatus > 0 AND fbRmtClprUnclampChk.udiStatus < 65534) THEN
							tylocalMagConv2Clp.Out.bFixClprClampCtrl	:= FALSE;
							tylocalMagConv2Clp.Out.bRmtClprClampCtrl	:= FALSE;
							tylocalMagConv2Clp.Out.bFixClprUnClampCtrl	:= FALSE;
							tylocalMagConv2Clp.Out.bRmtClprUnClampCtrl	:= FALSE;

							tylocalMagConv2Clp.Out.eStatus	:= Error;

							IF fbFixClprUnclampChk.udiStatus = 1504 OR fbRmtClprUnclampChk.udiStatus = 1504 THEN
								udiStatus	:= 10002;	//Clamper Clamp Sensor Off Time Out In Unclamp Check While Conveyor Initial With Clamper
							ELSIF fbFixClprUnclampChk.udiStatus = 1505 OR fbRmtClprUnclampChk.udiStatus = 1505 THEN
								udiStatus	:= 10003;	//Clamper Unclamp Sensor On Time Out In Unclamp Check While Conveyor Initial With Clamper
							ELSIF fbFixClprUnclampChk.udiStatus = 1508 OR fbRmtClprUnclampChk.udiStatus = 1508 THEN
								udiStatus	:= 10004;	//Clamper Unclamp Safety Sensor Error In Unclamp Check While Conveyor Initial With Clamper
							ELSE
								IF fbFixClprUnclampChk.udiStatus > 0 AND fbFixClprUnclampChk.udiStatus < 65534 THEN
									udiStatus	:= fbFixClprUnclampChk.udiStatus;
								ELSIF fbRmtClprUnclampChk.udiStatus > 0 AND fbRmtClprUnclampChk.udiStatus < 65534 THEN
									udiStatus	:= fbRmtClprUnclampChk.udiStatus;
								END_IF
							END_IF
						END_IF

					1:	//Conveyor Exit
						//Conveyor Run
						fbExit.bConvLToR	:= (tylocalMagConv2Clp.In.eDirection = ConvDirLToR) OR (tylocalMagConv2Clp.In.eDirection = ConvDirRToR);
						fbExit.tTimeOut		:= DINT_TO_TIME(tylocalMagConv2Clp.In.diTxOutTimeOut);

						IF fbExit.bConvLToR = TRUE THEN
							fbExit.bEndSen	:= tylocalMagConv2Clp.In.bRightSen;
						ELSE
							fbExit.bEndSen	:= tylocalMagConv2Clp.In.bLeftSen;
						END_IF

						fbExit(bEn := TRUE);

						tylocalMagConv2Clp.Out.bMtrSigOnOrLToR	:= fbExit.bMtrSigOnOrLToR;
						tylocalMagConv2Clp.Out.bMtrDirOrRToL	:= fbExit.bMtrDirOrRToL;

						IF fbExit.udiStatus = 0 THEN
							tylocalMagConv2Clp.Out.bHvMag		:= FALSE;
							tylocalMagConv2Clp.Out.eStatus		:= Done;
						ELSIF fbExit.udiStatus < 65534 THEN
							tylocalMagConv2Clp.Out.eStatus		:= Error;

							IF fbExit.udiStatus = 1101 THEN
								udiStatus	:= 10031;	//Transfer Out Time Out While Conveyor Exit With Clamper
							ELSE
								udiStatus	:= fbExit.udiStatus;
							END_IF
						END_IF

				END_CASE

			END_IF

		MagConv2ClpActExit1Clpr:
			IF tylocalMagConv2Clp.Out.eStatus = Idle OR tylocalMagConv2Clp.Out.eStatus = Busy THEN

				tylocalMagConv2Clp.Out.eStatus	:= Busy;

				CASE usiStep OF
					0:	//Unclamp
						tylocalMagConv2Clp.Out.bFixClprClampCtrl	:= FALSE;
						tylocalMagConv2Clp.Out.bRmtClprClampCtrl	:= FALSE;
						tylocalMagConv2Clp.Out.bFixClprUnClampCtrl := TRUE;
						tylocalMagConv2Clp.Out.bRmtClprUnClampCtrl	:= TRUE;

						fbFixClprUnclampChk.bExtSen		:= tylocalMagConv2Clp.In.bFixClprClampSen;
						fbFixClprUnclampChk.bRetSen		:= tylocalMagConv2Clp.In.bFixClprUnclampSen;
						fbFixClprUnclampChk.bRetSafety	:= tylocalMagConv2Clp.In.bFixClprUnclampSafetySen;
						fbFixClprUnclampChk(bEn := TRUE);

						fbRmtClprUnclampChk.bExtSen		:= tylocalMagConv2Clp.In.bRmtClprClampSen;
						fbRmtClprUnclampChk.bRetSen		:= tylocalMagConv2Clp.In.bRmtClprUnclampSen;
						fbRmtClprUnclampChk.bRetSafety	:= tylocalMagConv2Clp.In.bRmtClprUnclampSafetySen;
						fbRmtClprUnclampChk(bEn := TRUE);

						IF fbFixClprUnclampChk.udiStatus = 0 AND fbRmtClprUnclampChk.udiStatus = 0 THEN
							usiStep	:= 1;
						ELSIF (fbFixClprUnclampChk.udiStatus > 0 AND fbFixClprUnclampChk.udiStatus < 65534) OR (fbRmtClprUnclampChk.udiStatus > 0 AND fbRmtClprUnclampChk.udiStatus < 65534) THEN
							tylocalMagConv2Clp.Out.bFixClprClampCtrl	:= FALSE;
							tylocalMagConv2Clp.Out.bRmtClprClampCtrl	:= FALSE;
							tylocalMagConv2Clp.Out.bFixClprUnClampCtrl := FALSE;
							tylocalMagConv2Clp.Out.bRmtClprUnClampCtrl	:= FALSE;

							tylocalMagConv2Clp.Out.eStatus	:= Error;

							IF fbFixClprUnclampChk.udiStatus = 1504 OR fbRmtClprUnclampChk.udiStatus = 1504 THEN
								udiStatus	:= 10002;	//Clamper Clamp Sensor Off Time Out In Unclamp Check While Conveyor Initial With Clamper
							ELSIF fbFixClprUnclampChk.udiStatus = 1505 OR fbRmtClprUnclampChk.udiStatus = 1505 THEN
								udiStatus	:= 10003;	//Clamper Unclamp Sensor On Time Out In Unclamp Check While Conveyor Initial With Clamper
							ELSIF fbFixClprUnclampChk.udiStatus = 1508 OR fbRmtClprUnclampChk.udiStatus = 1508 THEN
								udiStatus	:= 10004;	//Clamper Unclamp Safety Sensor Error In Unclamp Check While Conveyor Initial With Clamper
							ELSE
								IF fbFixClprUnclampChk.udiStatus > 0 AND fbFixClprUnclampChk.udiStatus < 65534 THEN
									udiStatus	:= fbFixClprUnclampChk.udiStatus;
								ELSIF fbRmtClprUnclampChk.udiStatus > 0 AND fbRmtClprUnclampChk.udiStatus < 65534 THEN
									udiStatus	:= fbRmtClprUnclampChk.udiStatus;
								END_IF
							END_IF
						END_IF

					1:	//Conveyor Exit
						//Conveyor Run
						fbExit1.bConvLToR		:= (tylocalMagConv2Clp.In.eDirection = ConvDirLToR) OR (tylocalMagConv2Clp.In.eDirection = ConvDirRToR);
						fbExit1.tTimeOut		:= DINT_TO_TIME(tylocalMagConv2Clp.In.diTxOutTimeOut);

						IF fbExit1.bConvLToR = TRUE THEN
							fbExit1.bEndSen	:= tylocalMagConv2Clp.In.bRightSen;
						ELSE
							fbExit1.bEndSen	:= tylocalMagConv2Clp.In.bLeftSen;
						END_IF

						fbExit1(bEn := TRUE);

						tylocalMagConv2Clp.Out.bMtrSigOnOrLToR	:= fbExit1.bMtrSigOnOrLToR;
						tylocalMagConv2Clp.Out.bMtrDirOrRToL	:= fbExit1.bMtrDirOrRToL;

						IF fbExit1.udiStatus = 0 THEN
							tylocalMagConv2Clp.Out.bHvMag		:= FALSE;
							tylocalMagConv2Clp.Out.eStatus		:= Done;
						ELSIF fbExit1.udiStatus < 65534 THEN
							tylocalMagConv2Clp.Out.eStatus		:= Error;

							IF fbExit1.udiStatus = 1101 THEN
								udiStatus	:= 10033;	//Transfer Out Time Out While Conveyor Exit With Clamper
							ELSE
								udiStatus	:= fbExit1.udiStatus;
							END_IF
						END_IF

				END_CASE

			END_IF

		MagConv2ClpActFixClprSetAll:
			IF tylocalMagConv2Clp.Out.eStatus = Idle OR tylocalMagConv2Clp.Out.eStatus = Busy THEN

				tylocalMagConv2Clp.Out.eStatus	:= Busy;

				tylocalMagConv2Clp.Out.bMtrSigOnOrLToR	:= FALSE;
				tylocalMagConv2Clp.Out.bMtrDirOrRToL	:= FALSE;

				tylocalMagConv2Clp.Out.bFixClprClampCtrl	:= TRUE;
				tylocalMagConv2Clp.Out.bFixClprUnClampCtrl := TRUE;

				tylocalMagConv2Clp.Out.eStatus	:= Done;

			END_IF

		MagConv2ClpActFixClprRstAll:
			IF tylocalMagConv2Clp.Out.eStatus = Idle OR tylocalMagConv2Clp.Out.eStatus = Busy THEN

				tylocalMagConv2Clp.Out.eStatus	:= Busy;

				tylocalMagConv2Clp.Out.bMtrSigOnOrLToR	:= FALSE;
				tylocalMagConv2Clp.Out.bMtrDirOrRToL	:= FALSE;

				tylocalMagConv2Clp.Out.bFixClprClampCtrl	:= FALSE;
				tylocalMagConv2Clp.Out.bFixClprUnClampCtrl := FALSE;

				tylocalMagConv2Clp.Out.eStatus	:= Done;

			END_IF

		MagConv2ClpActFixClprSetClamp:
			IF tylocalMagConv2Clp.Out.eStatus = Idle OR tylocalMagConv2Clp.Out.eStatus = Busy THEN

				tylocalMagConv2Clp.Out.eStatus	:= Busy;

				tylocalMagConv2Clp.Out.bMtrSigOnOrLToR	:= FALSE;
				tylocalMagConv2Clp.Out.bMtrDirOrRToL	:= FALSE;

				tylocalMagConv2Clp.Out.bFixClprClampCtrl	:= TRUE;
				tylocalMagConv2Clp.Out.bFixClprUnClampCtrl := FALSE;

				tylocalMagConv2Clp.Out.eStatus	:= Done;

			END_IF

		MagConv2ClpActFixClprSetUnclamp:
			IF tylocalMagConv2Clp.Out.eStatus = Idle OR tylocalMagConv2Clp.Out.eStatus = Busy THEN

				tylocalMagConv2Clp.Out.eStatus	:= Busy;

				tylocalMagConv2Clp.Out.bMtrSigOnOrLToR	:= FALSE;
				tylocalMagConv2Clp.Out.bMtrDirOrRToL	:= FALSE;

				tylocalMagConv2Clp.Out.bFixClprClampCtrl	:= FALSE;
				tylocalMagConv2Clp.Out.bFixClprUnClampCtrl := TRUE;

				tylocalMagConv2Clp.Out.eStatus	:= Done;

			END_IF

		MagConv2ClpActFixClprClamp:
			IF tylocalMagConv2Clp.Out.eStatus = Idle OR tylocalMagConv2Clp.Out.eStatus = Busy THEN

				tylocalMagConv2Clp.Out.eStatus	:= Busy;

				tylocalMagConv2Clp.Out.bMtrSigOnOrLToR	:= FALSE;
				tylocalMagConv2Clp.Out.bMtrDirOrRToL	:= FALSE;

				tylocalMagConv2Clp.Out.bFixClprClampCtrl	:= TRUE;
				tylocalMagConv2Clp.Out.bFixClprUnClampCtrl := FALSE;

				fbFixClprClampChk.bExtSen		:= tylocalMagConv2Clp.In.bFixClprClampSen;
				fbFixClprClampChk.bRetSen		:= tylocalMagConv2Clp.In.bFixClprUnclampSen;
				fbFixClprClampChk.bExtSafety	:= tylocalMagConv2Clp.In.bFixClprClampSafetySen;
				fbFixClprClampChk(bEn := TRUE);

				IF fbFixClprClampChk.udiStatus = 0 THEN
					tylocalMagConv2Clp.Out.eStatus	:= Done;
				ELSIF fbFixClprClampChk.udiStatus < 65534 THEN
					tylocalMagConv2Clp.Out.bFixClprClampCtrl	:= FALSE;
					tylocalMagConv2Clp.Out.bFixClprUnClampCtrl := FALSE;

					tylocalMagConv2Clp.Out.eStatus	:= Error;

					IF fbFixClprClampChk.udiStatus = 1503 THEN
						udiStatus	:= 10016;	//Clamper Clamp Sensor On Time Out In Clamp Check While Clamper Clamp
					ELSIF fbFixClprClampChk.udiStatus = 1506 THEN
						udiStatus	:= 10017;	//Clamper Unclamp Sensor Off Time Out In Clamp Check While Clamper Clamp
					ELSIF fbFixClprClampChk.udiStatus = 1507 THEN
						udiStatus	:= 10018;	//Clamper Clamp Safety Sensor Error In Clamp Check While Clamper Clamp
					ELSE
						udiStatus	:= fbFixClprClampChk.udiStatus;
					END_IF
				END_IF
			END_IF

		MagConv2ClpActFixClprUnclamp:
			IF tylocalMagConv2Clp.Out.eStatus = Idle OR tylocalMagConv2Clp.Out.eStatus = Busy THEN

				tylocalMagConv2Clp.Out.eStatus	:= Busy;

				tylocalMagConv2Clp.Out.bMtrSigOnOrLToR	:= FALSE;
				tylocalMagConv2Clp.Out.bMtrDirOrRToL	:= FALSE;

				tylocalMagConv2Clp.Out.bFixClprClampCtrl	:= FALSE;
				tylocalMagConv2Clp.Out.bFixClprUnClampCtrl := TRUE;

				fbFixClprUnclampChk.bExtSen		:= tylocalMagConv2Clp.In.bFixClprClampSen;
				fbFixClprUnclampChk.bRetSen		:= tylocalMagConv2Clp.In.bFixClprUnclampSen;
				fbFixClprUnclampChk.bRetSafety	:= tylocalMagConv2Clp.In.bFixClprUnclampSafetySen;
				fbFixClprUnclampChk(bEn := TRUE);

				IF fbFixClprUnclampChk.udiStatus = 0 THEN
					tylocalMagConv2Clp.Out.eStatus	:= Done;
				ELSIF fbFixClprUnclampChk.udiStatus < 65534 THEN
					tylocalMagConv2Clp.Out.bFixClprClampCtrl	:= FALSE;
					tylocalMagConv2Clp.Out.bFixClprUnClampCtrl := FALSE;

					tylocalMagConv2Clp.Out.eStatus	:= Error;

					IF fbFixClprUnclampChk.udiStatus = 1504 THEN
						udiStatus	:= 10019;	//Clamper Clamp Sensor Off Time Out In Unclamp Check While Clamper Unclamp
					ELSIF fbFixClprUnclampChk.udiStatus = 1505 THEN
						udiStatus	:= 10020;	//Clamper Unclamp Sensor On Time Out In Unclamp Check While Clamper Unclamp
					ELSIF fbFixClprUnclampChk.udiStatus = 1508 THEN
						udiStatus	:= 10021;	//Clamper Unclamp Safety Sensor Error In Unclamp Check While Clamper Unclamp
					ELSE
						udiStatus	:= fbFixClprUnclampChk.udiStatus;
					END_IF
				END_IF

			END_IF

		MagConv2ClpActRmtClprSetAll:
			IF tylocalMagConv2Clp.Out.eStatus = Idle OR tylocalMagConv2Clp.Out.eStatus = Busy THEN

				tylocalMagConv2Clp.Out.eStatus	:= Busy;

				tylocalMagConv2Clp.Out.bMtrSigOnOrLToR	:= FALSE;
				tylocalMagConv2Clp.Out.bMtrDirOrRToL	:= FALSE;

				tylocalMagConv2Clp.Out.bRmtClprClampCtrl	:= TRUE;
				tylocalMagConv2Clp.Out.bRmtClprUnClampCtrl	:= TRUE;
				tylocalMagConv2Clp.Out.eStatus	:= Done;

			END_IF

		MagConv2ClpActRmtClprRstAll:
			IF tylocalMagConv2Clp.Out.eStatus = Idle OR tylocalMagConv2Clp.Out.eStatus = Busy THEN

				tylocalMagConv2Clp.Out.eStatus	:= Busy;

				tylocalMagConv2Clp.Out.bMtrSigOnOrLToR	:= FALSE;
				tylocalMagConv2Clp.Out.bMtrDirOrRToL	:= FALSE;

				tylocalMagConv2Clp.Out.bRmtClprClampCtrl	:= FALSE;
				tylocalMagConv2Clp.Out.bRmtClprUnClampCtrl	:= FALSE;
				tylocalMagConv2Clp.Out.eStatus	:= Done;

			END_IF

		MagConv2ClpActRmtClprSetClamp:
			IF tylocalMagConv2Clp.Out.eStatus = Idle OR tylocalMagConv2Clp.Out.eStatus = Busy THEN

				tylocalMagConv2Clp.Out.eStatus	:= Busy;

				tylocalMagConv2Clp.Out.bMtrSigOnOrLToR	:= FALSE;
				tylocalMagConv2Clp.Out.bMtrDirOrRToL	:= FALSE;

				tylocalMagConv2Clp.Out.bRmtClprClampCtrl	:= TRUE;
				tylocalMagConv2Clp.Out.bRmtClprUnClampCtrl	:= FALSE;
				tylocalMagConv2Clp.Out.eStatus	:= Done;

			END_IF

		MagConv2ClpActRmtClprSetUnclamp:
			IF tylocalMagConv2Clp.Out.eStatus = Idle OR tylocalMagConv2Clp.Out.eStatus = Busy THEN

				tylocalMagConv2Clp.Out.eStatus	:= Busy;

				tylocalMagConv2Clp.Out.bMtrSigOnOrLToR	:= FALSE;
				tylocalMagConv2Clp.Out.bMtrDirOrRToL	:= FALSE;

				tylocalMagConv2Clp.Out.bRmtClprClampCtrl	:= FALSE;
				tylocalMagConv2Clp.Out.bRmtClprUnClampCtrl	:= TRUE;

				tylocalMagConv2Clp.Out.eStatus	:= Done;

			END_IF

		MagConv2ClpActRmtClprClamp:
			IF tylocalMagConv2Clp.Out.eStatus = Idle OR tylocalMagConv2Clp.Out.eStatus = Busy THEN

				tylocalMagConv2Clp.Out.eStatus	:= Busy;

				tylocalMagConv2Clp.Out.bMtrSigOnOrLToR	:= FALSE;
				tylocalMagConv2Clp.Out.bMtrDirOrRToL	:= FALSE;

				tylocalMagConv2Clp.Out.bRmtClprClampCtrl	:= TRUE;
				tylocalMagConv2Clp.Out.bRmtClprUnClampCtrl	:= FALSE;

				fbRmtClprClampChk.bExtSen		:= tylocalMagConv2Clp.In.bRmtClprClampSen;
				fbRmtClprClampChk.bRetSen		:= tylocalMagConv2Clp.In.bRmtClprUnclampSen;
				fbRmtClprClampChk.bExtSafety	:= tylocalMagConv2Clp.In.bRmtClprClampSafetySen;
				fbRmtClprClampChk(bEn := TRUE);

				IF fbRmtClprClampChk.udiStatus = 0 THEN
					tylocalMagConv2Clp.Out.eStatus	:= Done;
				ELSIF fbRmtClprClampChk.udiStatus < 65534 THEN
					tylocalMagConv2Clp.Out.bRmtClprClampCtrl	:= FALSE;
					tylocalMagConv2Clp.Out.bRmtClprUnClampCtrl	:= FALSE;
					tylocalMagConv2Clp.Out.eStatus	:= Error;

					IF fbRmtClprClampChk.udiStatus = 1503 THEN
						udiStatus	:= 10016;	//Clamper Clamp Sensor On Time Out In Clamp Check While Clamper Clamp
					ELSIF fbRmtClprClampChk.udiStatus = 1506 THEN
						udiStatus	:= 10017;	//Clamper Unclamp Sensor Off Time Out In Clamp Check While Clamper Clamp
					ELSIF fbRmtClprClampChk.udiStatus = 1507 THEN
						udiStatus	:= 10018;	//Clamper Clamp Safety Sensor Error In Clamp Check While Clamper Clamp
					ELSE
						udiStatus	:= fbRmtClprClampChk.udiStatus;
					END_IF
				END_IF
			END_IF

		MagConv2ClpActRmtClprUnclamp:
			IF tylocalMagConv2Clp.Out.eStatus = Idle OR tylocalMagConv2Clp.Out.eStatus = Busy THEN

				tylocalMagConv2Clp.Out.eStatus	:= Busy;

				tylocalMagConv2Clp.Out.bMtrSigOnOrLToR	:= FALSE;
				tylocalMagConv2Clp.Out.bMtrDirOrRToL	:= FALSE;

				tylocalMagConv2Clp.Out.bRmtClprClampCtrl	:= FALSE;
				tylocalMagConv2Clp.Out.bRmtClprUnClampCtrl	:= TRUE;

				fbRmtClprUnclampChk.bExtSen		:= tylocalMagConv2Clp.In.bRmtClprClampSen;
				fbRmtClprUnclampChk.bRetSen		:= tylocalMagConv2Clp.In.bRmtClprUnclampSen;
				fbRmtClprUnclampChk.bRetSafety	:= tylocalMagConv2Clp.In.bRmtClprUnclampSafetySen;
				fbRmtClprUnclampChk(bEn := TRUE);

				IF fbRmtClprUnclampChk.udiStatus = 0 THEN
					tylocalMagConv2Clp.Out.eStatus	:= Done;
				ELSIF fbRmtClprUnclampChk.udiStatus < 65534 THEN
					tylocalMagConv2Clp.Out.bRmtClprClampCtrl	:= FALSE;
					tylocalMagConv2Clp.Out.bRmtClprUnClampCtrl	:= FALSE;
					tylocalMagConv2Clp.Out.eStatus	:= Error;

					IF fbRmtClprUnclampChk.udiStatus = 1504 THEN
						udiStatus	:= 10019;	//Clamper Clamp Sensor Off Time Out In Unclamp Check While Clamper Unclamp
					ELSIF fbRmtClprUnclampChk.udiStatus = 1505 THEN
						udiStatus	:= 10020;	//Clamper Unclamp Sensor On Time Out In Unclamp Check While Clamper Unclamp
					ELSIF fbRmtClprUnclampChk.udiStatus = 1508 THEN
						udiStatus	:= 10021;	//Clamper Unclamp Safety Sensor Error In Unclamp Check While Clamper Unclamp
					ELSE
						udiStatus	:= fbRmtClprUnclampChk.udiStatus;
					END_IF
				END_IF

			END_IF

		MagConv2ClpActStop:
			IF tylocalMagConv2Clp.Out.eStatus = Idle OR tylocalMagConv2Clp.Out.eStatus = Busy THEN

				tylocalMagConv2Clp.Out.eStatus	:= Busy;

				//Conveyor Run
				fbStop(bEn := TRUE);

				tylocalMagConv2Clp.Out.bMtrSigOnOrLToR	:= fbStop.bMtrSigOnOrLToR;
				tylocalMagConv2Clp.Out.bMtrDirOrRToL	:= fbStop.bMtrDirOrRToL;

				IF fbStop.udiStatus = 0 THEN
					tylocalMagConv2Clp.Out.eStatus	:= Done;
				ELSIF fbStop.udiStatus < 65534 THEN
					udiStatus	:= fbStop.udiStatus;
					tylocalMagConv2Clp.Out.eStatus		:= Error;
				END_IF

			END_IF

		MagConv2ClpActStopClpr:
			IF tylocalMagConv2Clp.Out.eStatus = Idle OR tylocalMagConv2Clp.Out.eStatus = Busy THEN

				tylocalMagConv2Clp.Out.eStatus	:= Busy;

				//Conveyor Run
				fbStop(bEn := TRUE);

				tylocalMagConv2Clp.Out.bMtrSigOnOrLToR	:= fbStop.bMtrSigOnOrLToR;
				tylocalMagConv2Clp.Out.bMtrDirOrRToL	:= fbStop.bMtrDirOrRToL;

				tylocalMagConv2Clp.Out.bFixClprClampCtrl	:= FALSE;
				tylocalMagConv2Clp.Out.bRmtClprClampCtrl	:= FALSE;
				tylocalMagConv2Clp.Out.bFixClprUnClampCtrl := TRUE;
				tylocalMagConv2Clp.Out.bRmtClprUnClampCtrl	:= TRUE;

				fbFixClprUnclampChk.bExtSen		:= tylocalMagConv2Clp.In.bFixClprClampSen;
				fbFixClprUnclampChk.bRetSen		:= tylocalMagConv2Clp.In.bFixClprUnclampSen;
				fbFixClprUnclampChk.bRetSafety	:= tylocalMagConv2Clp.In.bFixClprUnclampSafetySen;
				fbFixClprUnclampChk(bEn := TRUE);

				fbRmtClprUnclampChk.bExtSen		:= tylocalMagConv2Clp.In.bRmtClprClampSen;
				fbRmtClprUnclampChk.bRetSen		:= tylocalMagConv2Clp.In.bRmtClprUnclampSen;
				fbRmtClprUnclampChk.bRetSafety	:= tylocalMagConv2Clp.In.bRmtClprUnclampSafetySen;
				fbRmtClprUnclampChk(bEn := TRUE);

				IF fbStop.udiStatus = 0 AND fbFixClprUnclampChk.udiStatus = 0 AND fbRmtClprUnclampChk.udiStatus = 0 THEN
					tylocalMagConv2Clp.Out.eStatus		:= Done;
				ELSIF fbStop.udiStatus > 0 AND fbStop.udiStatus < 65534 THEN
					udiStatus	:= fbStop.udiStatus;
					tylocalMagConv2Clp.Out.eStatus		:= Error;
				ELSIF (fbFixClprUnclampChk.udiStatus > 0 AND fbFixClprUnclampChk.udiStatus < 65534) OR (fbRmtClprUnclampChk.udiStatus > 0 AND fbRmtClprUnclampChk.udiStatus < 65534) THEN
					tylocalMagConv2Clp.Out.bFixClprClampCtrl	:= FALSE;
					tylocalMagConv2Clp.Out.bRmtClprClampCtrl	:= FALSE;
					tylocalMagConv2Clp.Out.bFixClprUnClampCtrl := FALSE;
					tylocalMagConv2Clp.Out.bRmtClprUnClampCtrl	:= FALSE;

					tylocalMagConv2Clp.Out.eStatus	:= Error;

					IF fbFixClprUnclampChk.udiStatus = 1504 OR fbRmtClprUnclampChk.udiStatus = 1504 THEN
						udiStatus	:= 10022;	//Clamper Clamp Sensor Off Time Out In Unclamp Check While Stop With Clamper
					ELSIF fbFixClprUnclampChk.udiStatus = 1505 OR fbRmtClprUnclampChk.udiStatus = 1505 THEN
						udiStatus	:= 10023;	//Clamper Unclamp Sensor On Time Out In Unclamp Check While Stop With Clamper
					ELSIF fbFixClprUnclampChk.udiStatus = 1508 OR fbRmtClprUnclampChk.udiStatus = 1508 THEN
						udiStatus	:= 10024;	//Clamper Unclamp Safety Sensor Error In Unclamp Check While Stop With Clamper
					ELSE
						IF fbFixClprUnclampChk.udiStatus > 0 AND fbFixClprUnclampChk.udiStatus < 65534 THEN
							udiStatus	:= fbFixClprUnclampChk.udiStatus;
						ELSIF fbRmtClprUnclampChk.udiStatus > 0 AND fbRmtClprUnclampChk.udiStatus < 65534 THEN
							udiStatus	:= fbRmtClprUnclampChk.udiStatus;
						END_IF
					END_IF
				END_IF

			END_IF

		MagConv2ClpActSetMtrSigOnOrLToR:
			IF tylocalMagConv2Clp.Out.eStatus = Idle OR tylocalMagConv2Clp.Out.eStatus = Busy THEN

				tylocalMagConv2Clp.Out.bMtrSigOnOrLToR	:= TRUE;

				tylocalMagConv2Clp.Out.eStatus	:= Done;

			END_IF

		MagConv2ClpActSetMtrDirOrRToL:
			IF tylocalMagConv2Clp.Out.eStatus = Idle OR tylocalMagConv2Clp.Out.eStatus = Busy THEN

				tylocalMagConv2Clp.Out.bMtrDirOrRToL	:= TRUE;

				tylocalMagConv2Clp.Out.eStatus	:= Done;

			END_IF

		MagConv2ClpActRstMtrSigOnOrLToR:
			IF tylocalMagConv2Clp.Out.eStatus = Idle OR tylocalMagConv2Clp.Out.eStatus = Busy THEN

				tylocalMagConv2Clp.Out.bMtrSigOnOrLToR	:= FALSE;

				tylocalMagConv2Clp.Out.eStatus	:= Done;

			END_IF

		MagConv2ClpActRstMtrDirOrRToL:
			IF tylocalMagConv2Clp.Out.eStatus = Idle OR tylocalMagConv2Clp.Out.eStatus = Busy THEN

				tylocalMagConv2Clp.Out.bMtrDirOrRToL	:= FALSE;

				tylocalMagConv2Clp.Out.eStatus	:= Done;

			END_IF

		MagConv2ClpActSetMtrAll:
			IF tylocalMagConv2Clp.Out.eStatus = Idle OR tylocalMagConv2Clp.Out.eStatus = Busy THEN

				tylocalMagConv2Clp.Out.bMtrSigOnOrLToR	:= TRUE;
				tylocalMagConv2Clp.Out.bMtrDirOrRToL	:= TRUE;

				tylocalMagConv2Clp.Out.eStatus	:= Done;

			END_IF

		MagConv2ClpActRstMtrAll:
			IF tylocalMagConv2Clp.Out.eStatus = Idle OR tylocalMagConv2Clp.Out.eStatus = Busy THEN

				tylocalMagConv2Clp.Out.bMtrSigOnOrLToR	:= FALSE;
				tylocalMagConv2Clp.Out.bMtrDirOrRToL	:= FALSE;

				tylocalMagConv2Clp.Out.eStatus	:= Done;

			END_IF

	END_CASE

END_ACTION
```

#### Act_Alarm.st - Do Not Change!!!
```iecst
(** 2019-10-30 **)
ACTION Act_Alarm:

	//Error
	IF EDGEPOS(eStatus = Error) THEN

		tyAlmData.sProgNm		:= p_sProgNm;
		tyAlmData.udiCode		:= udiStatus;
		tyAlmData.eSeverity		:= AlmSeverityError;
		tyAlmData.udiRunTime	:= tyAlmData.udiRunTime + 1;
		tyAlmData.bAlm			:= TRUE;
		tyAlmData.udiModuleNum  := udiModuleNum;
		g_sMagConv2ClpProgNm		:= p_sProgNm;

		//Get Error Message
		IF tyAlmData.udiCode < 10000 OR tyAlmData.udiCode > 10099 THEN
			tyAlmData.sAlmMsg	:= 'Unknown';
			tyAlmData.sRcyMsg	:= 'Unknown';
		ELSE
			tyAlmData.sAlmMsg	:= a_tyAlmText[tyAlmData.udiCode].sAlmText;
			tyAlmData.sRcyMsg	:= a_tyAlmText[tyAlmData.udiCode].sRcyText;
		END_IF

		sStatTxt	:= tyAlmData.sAlmMsg;

	ELSIF bRstErr AND (tyAlmData.udiCode <> 0) THEN

		tyAlmData.udiCode	:= 0;
		tyAlmData.eSeverity	:= AlmSeverityNA;
		tyAlmData.sAlmMsg	:= '';
		tyAlmData.sRcyMsg	:= '';
		tyAlmData.bAlm			:= FALSE;
		sStatTxt	:= a_sStatText[eStat];

	END_IF

END_ACTION
```

#### Local.var - Do Not Change!!!
```iecst
(*2019-10-30*)
VAR
	tylocalMagConv2Clp : tyMagConv2Clp;
END_VAR
(**)
(*Local Action, State & Status*)
VAR
	eAct : eMagConv2ClpAction := MagConv2ClpActIdle;
	udiStatus : UDINT := 0;
	a_sStatText : ARRAY[0..50] OF STRING[200] := ['Idling','Initializing','Initializing With Stop Then Clamper','Initializing With Clamper Then Stop','Entering Board','Entering Board With Stop Then Clamper','Entering Board With Clamper Then Stop','Pre-Exiting Board','Pre-Exiting Board With Clamper',2('Exiting Board'),2('Exiting Board With Clamper'),'Fix/Bottom Clamper Setting All Control','Fix/Bottom Clamper Resetting All Control','Fix/Bottom Clamper Setting Clamp','Fix/Bottom Clamper Setting Unclamp','Fix/Bottom Clamper Clamp','Fix/Bottom Clampler Unclamp','Remote/Top Clamper Setting All Control','Remote/Top Clamper Resetting All Control','Remote/Top Clamper Setting Clamp','Remote/Top Clamper Setting Unclamp','Remote/Top Clamper Clamp','Remote/Top Clampler Unclamp','Stopping','Stopping With Clamper','Turning On Motor Signal','Turning On Motor Direction','Turning Off Motor Signal','Turning Off Motor Direction','Turning On All Motor Output','Turning Off All Motor Output',18('')];
END_VAR
(**)
(*Local Alarm*)
VAR
	tyAlmData : tyAlmDat;
END_VAR
(**)
(*Local Output*)
VAR
	bHvMag : BOOL := FALSE;
	bMtrSigOnOrLToR : BOOL := FALSE;
	bMtrDirOrRToL : BOOL := FALSE;
	bFixClprClampCtrl : BOOL;
	bRmtClprClampCtrl : BOOL;
	bClprTwoOutputControl : BOOL := FALSE;
END_VAR
(**)
(*Local Input*)
VAR
	udiRstErr : UDINT := 0;
	bPrep : BOOL := TRUE;
	bEn : BOOL := TRUE;
	bDis : BOOL := FALSE;
	bManual : BOOL := FALSE;
	bOnDirMod : BOOL := FALSE;
	diInitTm : DINT := 10000;
	tMtrOffDlyTm : TIME := T#0S;
	diTxInTimeOut : DINT := 10000;
	diTxOutTimeOut : DINT := 10000;
	eDirection : eConvDir := ConvDirLToR;
	bLeftSen : BOOL := FALSE;
	bRightSen : BOOL := FALSE;
	bFixClprClampSen : BOOL := FALSE;
	bFixClprUnclampSen : BOOL := FALSE;
	bFixClprClampSafetySen : BOOL := TRUE;
	bFixClprUnclampSafetySen : BOOL := TRUE;
	bRmtClprClampSen : BOOL := FALSE;
	bRmtClprUnclampSen : BOOL := FALSE;
	bRmtClprClampSafetySen : BOOL := TRUE;
	bRmtClprUnclampSafetySen : BOOL := TRUE;
	bWidthChkPrep : BOOL := TRUE;
	sProgNm : STRING[15] := 'MagConv2Clp';
	tClprClampTO : TIME := T#20s;
	tClprUnclampTO : TIME := T#20s;
	bNtSettingsLoadDone : BOOL := TRUE;
END_VAR
(**)
(*Local*)
VAR
	bRstErr : BOOL;
	udiRstErrOld : UDINT;
	bInitDone : BOOL;
	bInitialDone : BOOL;
	bReachEnd : BOOL;
	usiStep : USINT;
	usiSubStep : USINT;
	eStatOld : eMagConv2ClpAction := MagConv2ClpActIdle;
	fbInit : fbConvSenToSenTm;
	fbEnt : fbConvSenToSen;
	fbPreExit : fbConvSenToSenTm;
	fbExit : fbConvSenToSenOff;
	fbExit1 : fbConvSenToSenOff1;
	fbStop : fbConvMtrOff;
	fbFixClprClampChk : fbPneuExtRetSenExtChk;
	fbFixClprUnclampChk : fbPneuExtRetSenRetChk;
	fbRmtClprClampChk : fbPneuExtRetSenExtChk;
	fbFixClprDly : TON := (PT:=T#1s);
	fbRmtClprUnclampChk : fbPneuExtRetSenRetChk;
	fbClprDlyTm : TON;
	fbSmallLargeSenDlyTm : TON := (PT:=T#1S);
	fbWidthChk : TON := (PT:=T#30s);
	fbLeftSenDelayTm : TON := (PT:=T#1S);
	fbFixClpExtChkTm : TON := (PT:=T#5s);
	fbRmtClpExtChkTm : TON := (PT:=T#3s);
	udiModuleNum : UDINT := 1901;
END_VAR
```

#### Act_InputConfig.st - not listed in the package file held
```iecst
(** 2019-10-30 **)
ACTION Act_InputConfig:

	(* Always Change If Project Change *)

	//Pass Data To Link

	tylocalMagConv2Clp.In.bLinkDISafetyRlySig := g_tyDInput.bSafetyRlySig;

	tylocalMagConv2Clp.In.bLinkMagSmallSen := g_tyDInput.bMagConvSmallMagSen3;
	tylocalMagConv2Clp.In.bLinkMagLargeSen := g_tyDInput.bMagConvLargeMagSen3;
	tylocalMagConv2Clp.In.bLinkFixClprUnClampSen := g_tyDInput.bMag3FixedUnclampRS;
	//	tylocalMagConv2Clp.In.bLinkFixClprClampSen := g_tyDInput.bMag3FixedClampRS; // Pneumatic Clamp Reed Switch
	tylocalMagConv2Clp.In.bLinkFixClprMagDetectSen := g_tyDInput.bMag3FixedClampSen; // Clamping Done Before Pneumatic Clamp Reed Switch for special Condition
	tylocalMagConv2Clp.In.bLinkFixClprMagDetectSenPrep := g_tyNtParamCurr.bProjFixClpMagDSenPrep; // Fixed Clamp Detect Sensor Prep before Clamp RS

	tylocalMagConv2Clp.In.bLinkMagOpsStepMagFullExit := g_tyOpsMagConvUL3MagFullExit;
	tylocalMagConv2Clp.In.bLinkDIMagEntSen := g_tyDInput.bMagConvEntSen3;
	//	tylocalMagConv2Clp.In.bLinkDO := g_tyDO;

	tylocalMagConv2Clp.In.bWidthChkSen := g_tyNtParamCurr.bCurtainSenPrep;
	tylocalMagConv2Clp.In.bWidthChkInterrupt := g_tyDInput.bCurtainSen;

	tylocalMagConv2Clp.In.bLinkNtParamMagModelAutoVerify := g_tyNtParamCurr.bProjMagAutoVerifyPrep;
	//	tylocalMagConv2Clp.In.tyDISettings := g_tyNtParamCurr.tyDISettings;
	//	tylocalMagConv2Clp.In.bLinkFixClprClampSen ACCESS ADR(bFixClprClampSen);//tylocalMagConv2Clp.In.DIMag1FixedSideDetect;//tylocalMagConv2Clp.In.DIMag1FixedClampRS; //initLocal at 1st

	//Pass Data To Internal Use
	tylocalMagConv2Clp.In.udiRstErr := g_tyRstErrReset;
	tylocalMagConv2Clp.In.bPrep := g_tyNtParamCurr.bProjMag3ConvPrep;
	tylocalMagConv2Clp.In.bManual := g_tyUIMnlMod;
	tylocalMagConv2Clp.In.bOnDirMod := g_tyNtParamCurr.bMagConv3OnDirMod;
	tylocalMagConv2Clp.In.diInitTm := g_tyMcParamCurr.tMag3ConvRunTmOut;
	tylocalMagConv2Clp.In.tMtrOffDlyTm := g_tyNtParamCurr.tMagConv3MtrOffDlyTm;
	tylocalMagConv2Clp.In.diTxInTimeOut := g_tyMcParamCurr.tMag3ConvRunTmOut;
	tylocalMagConv2Clp.In.diTxOutTimeOut := g_tyMcParamCurr.tMag3ConvRunTmOut;
	tylocalMagConv2Clp.In.eDirection := g_tyNtParamCurr.bProjMagConvDir;
	tylocalMagConv2Clp.In.sProgNm := g_tyNtParamCurr.sMagConv3ProgNm;
	tylocalMagConv2Clp.In.tClprClampTO := g_tyNtParamCurr.tMagConv3ClprClampTO;
	tylocalMagConv2Clp.In.tClprUnclampTO := g_tyNtParamCurr.tMagConv3ClprUnclampTO;
	//	tylocalMagConv2Clp.In.bLeftSen := g_tyDInput.bMagPresentSen3;
	tylocalMagConv2Clp.In.bRightSen	:= g_tyDInput.bMagPresentSen3;

	(* Always Change If Project Change *)

	IF g_tyOps.bRun THEN
		tylocalMagConv2Clp.In.eAct := g_tyOpsMagConvUL3.eMagConv2ClpAct;
	ELSIF tylocalMagConv2Clp.In.bManual = TRUE THEN
		tylocalMagConv2Clp.In.eAct := g_tyUIOut.eMnlAct.eMagConv2Clp3Act;
	ELSE
		tylocalMagConv2Clp.In.eAct := eAct;
	END_IF
	END_ACTION
```

#### Act_OutputConfig.st - not listed in the package file held
```iecst
ACTION Act_OutputConfig:
	// Output: Assign To Global For Independent Package Usage

	g_tyPneuMag3AWEngage := tylocalMagConv3Clp.Out; // Change the Global Naming According to the Physical Hardware Module

END_ACTION
```

### MagConv2Clp1.var - not listed in the package file held
```iecst
(*2019-10-30*)
(**)
(*Action & State & Status*)
VAR
	p_MagConv2Clp1Stat : UDINT;
	p_MagConv2Clp1Status : UDINT;
	p_MagConv2Clp1StatTxt : UDINT;
END_VAR
(**)
(*Alarm*)
VAR
	p_MagConv2Clp1AlmData : UDINT;
END_VAR
(**)
(*Output*)
VAR
	p_MagConv2Clp1HvMag : UDINT;
	p_MagConv2Clp1MtrSigOnOrLToR : UDINT;
	p_MagConv2Clp1MtrDirOrRToL : UDINT;
	p_MagConv2Clp1FixClprClampCtrl : UDINT;
	p_MagConv2Clp1RmtClprClampCtrl : UDINT;
	p_MagConv2Clp1ClprTwoOutputCtrl : UDINT;
END_VAR
```

### MagConv2Clp2.var - not listed in the package file held
```iecst
(*2019-10-30*)
(**)
(*Action & State & Status*)
VAR
	p_MagConv2Clp2Stat : UDINT;
	p_MagConv2Clp2Status : UDINT;
	p_MagConv2Clp2StatTxt : UDINT;
END_VAR
(**)
(*Alarm*)
VAR
	p_MagConv2Clp2AlmData : UDINT;
END_VAR
(**)
(*Output*)
VAR
	p_MagConv2Clp2HvMag : UDINT;
	p_MagConv2Clp2MtrSigOnOrLToR : UDINT;
	p_MagConv2Clp2MtrDirOrRToL : UDINT;
	p_MagConv2Clp2FixClprClampCtrl : UDINT;
	p_MagConv2Clp2RmtClprClampCtrl : UDINT;
	p_MagConv2Clp2ClprTwoOutputCtrl : UDINT;
END_VAR
```

### MagConv2Clp3.var - not listed in the package file held
```iecst
(*2019-10-30*)
(**)
(*Action & State & Status*)
VAR
	p_MagConv2Clp3Stat : UDINT;
	p_MagConv2Clp3Status : UDINT;
	p_MagConv2Clp3StatTxt : UDINT;
END_VAR
(**)
(*Alarm*)
VAR
	p_MagConv2Clp3AlmData : UDINT;
END_VAR
(**)
(*Output*)
VAR
	p_MagConv2Clp3HvMag : UDINT;
	p_MagConv2Clp3MtrSigOnOrLToR : UDINT;
	p_MagConv2Clp3MtrDirOrRToL : UDINT;
	p_MagConv2Clp3FixClprClampCtrl : UDINT;
	p_MagConv2Clp3RmtClprClampCtrl : UDINT;
	p_MagConv2Clp3ClprTwoOutputCtrl : UDINT;
END_VAR
```

### Conv.typ - Change By Project
```iecst
(*2019-06-17*)
(**)
(*Action*)

TYPE
	eConvAction :
		(
		ConvActIdle,
		ConvActInit,
		ConvActInitRev,
		ConvActInitPshr,
		ConvActInitPuller,
		ConvActInitRej,
		ConvActInitInsp,
		ConvActEnt,
		ConvActEntToInOff,
		ConvActEntRev,
		ConvActRev,
		ConvActRevImmedStart,
		ConvActEntPuller,
		ConvActEntRej,
		ConvActEntInsp,
		ConvActPreExit,
		ConvActRejResume,
		ConvActExit,
		ConvActExit1,
		ConvActExitPshr,
		ConvActExit1Pshr,
		ConvActPshrSetAll,
		ConvActPshrRstAll,
		ConvActPshrSetExt,
		ConvActPshrSetRet,
		ConvActPshrExt,
		ConvActPshrRet,
		ConvActPullerSetAll,
		ConvActPullerRstAll,
		ConvActPullerSetExt,
		ConvActPullerSetRet,
		ConvActPullerExt,
		ConvActPullerRet,
		ConvActRotSetAll,
		ConvActRotRstAll,
		ConvActRotSetHome,
		ConvActRotSetRmt,
		ConvActRotHome,
		ConvActRotRemote,
		ConvActRejSetAll,
		ConvActRejRstAll,
		ConvActRejSetUp,
		ConvActRejSetDown,
		ConvActRejUp,
		ConvActRejDown,
		ConvActStop,
		ConvActStopPshr,
		ConvActStopPuller,
		ConvActStopRej,
		ConvActSetMtrSigOnOrLToR,
		ConvActSetMtrDirOrRToL,
		ConvActRstMtrSigOnOrLToR,
		ConvActRstMtrDirOrRToL,
		ConvActSetMtrAll,
		ConvActRstMtrAll
		);
END_TYPE

(**)

TYPE
	eConvDir :
		(
		ConvDirLToR,
		ConvDirRToL,
		ConvDirLToL,
		ConvDirRToR
		);
END_TYPE

(**)

TYPE
	tyPshrConv : 	STRUCT
		In : tyPshrConvIn1;
		Out : tyPshrConvOut1;
	END_STRUCT;
	tyPshrConvIn1 : 	STRUCT
		eAct : eConvAction;
		udiRstErr : UDINT;
		bPrep : BOOL;
		bEn : BOOL;
		bDis : BOOL;
		bManual : BOOL;
		bLongBrdPrep : BOOL;
		bLongBrdEn : BOOL;
		bOnDirMod : BOOL;
		diInitTm : DINT;
		diRevDlyTm : DINT;
		tMtrOffDlyTm : TIME;
		diTxInTimeOut : DINT;
		diTxOutTimeOut : DINT;
		eDirection : eConvDir;
		bGdBrdInit : BOOL;
		bGdBrdEnt : BOOL;
		sProgNm : STRING[15];
		tPshrExtTO : TIME;
		tPshrRetTO : TIME;
		tPullerExtTO : TIME;
		tPullerRetTO : TIME;
		tRotHomeTO : TIME;
		tRotRemoteTO : TIME;
		tRejectUpTO : TIME;
		tRejectDownTO : TIME;
		bNtSettingsLoadDone : BOOL;
		bLeftSen : BOOL;
		bRightSen : BOOL;
		bMiddleSen : BOOL;
		bPullerChkSen : BOOL;
		bPshrExtSen : BOOL;
		bPshrRetSen : BOOL;
		bPshrExtSafetySen : BOOL;
		bPshrRetSafetySen : BOOL;
		bPullerExtSen : BOOL;
		bPullerRetSen : BOOL;
		bPullerExtSafetySen : BOOL;
		bPullerRetSafetySen : BOOL;
		bRotHomeSen : BOOL;
		bRotRemoteSen : BOOL;
		bRotHomeSafetySen : BOOL;
		bRotRemoteSafetySen : BOOL;
		bRejectUpSen : BOOL;
		bRejectDownSen : BOOL;
		bRejectUpSafetySen : BOOL;
		bRejectDownSafetySen : BOOL;
		bSelfTest : BOOL;
		bNtParamAutoRcpPrep : BOOL;
		bMcParamAutoRcpDis : BOOL;
		bLinkUIBypsInitConv : BOOL;
		bLinkDISafetyRlySig : BOOL;
		bLinkDIRgtSen : BOOL;
		bLinkDIClrSen : BOOL;
		usiLinkMcParamProdSelMcMod : USINT;
		eLinkOpsTravLifPosGo : eTravLifULPos;
		eLinkMcParamUSCommAMod : eMcSetCommMod;
		eLinkMcParamUSCommBMod : eMcSetCommMod;
		bLinkPshrRetSen : BOOL;
		bLinkPshrRetSlwSen : BOOL;
	END_STRUCT;
	tyPshrConvOut1 : 	STRUCT
		eStat : eConvAction;
		eStatus : eFBStatus;
		sStatTxt : STRING[200];
		tyAlmData : tyAlmDat;
		bHvBrd : BOOL;
		bRejHvBrd : BOOL;
		bInspHvBrd : BOOL;
		bGdBrd : BOOL;
		bLmtSenActivated : BOOL;
		bMtrSigOnOrLToR : BOOL;
		bMtrDirOrRToL : BOOL;
		bPshrExtCtrl : BOOL;
		bPshrRetCtrl : BOOL;
		bPshrTwoOutputControl : BOOL := FALSE;
		bPshrExtended : BOOL;
		bPshrRetracted : BOOL;
		bPullerExtCtrl : BOOL;
		bPullerRetCtrl : BOOL;
		bPullerTwoOutputControl : BOOL := TRUE;
		bPullerExtended : BOOL;
		bPullerRetracted : BOOL;
		bRotRemoteCtrl : BOOL;
		bRotTwoOutputControl : BOOL := FALSE;
		bRotAtRemote : BOOL;
		bRotAtHome : BOOL;
		bRejectUpCtrl : BOOL;
		bRejectDownCtrl : BOOL;
		bRejectTwoOutputControl : BOOL := TRUE;
		bRejectAtUp : BOOL;
		bRejectAtDown : BOOL;
		bPshrRetAllwTraverse : BOOL;
	END_STRUCT;
END_TYPE
```

### PshrConv.var - Change By Project
```iecst
(*2019-03-25*)
VAR
	g_tyPshrConv : tyPshrConvOut1;
END_VAR
```

### Program Logical/Conv/PshrConv (IEC) - 1.00.0 - NtConv v5.00.0 , NtPneu v5.00.0

#### InputRef.var
```iecst
(*2019-03-25*)
(**)
(*General*)
VAR
	p_eAct : REFERENCE TO eConvAction;
	p_udiRstErr : REFERENCE TO UDINT;
	p_bPrep : REFERENCE TO BOOL;
	p_bEn : REFERENCE TO BOOL;
	p_bDis : REFERENCE TO BOOL;
END_VAR
(**)
(*Configuration*)
VAR
	p_bManual : REFERENCE TO BOOL;
	p_bLongBrdPrep : REFERENCE TO BOOL;
	p_bLongBrdEn : REFERENCE TO BOOL;
	p_bOnDirMod : REFERENCE TO BOOL;
	p_diInitTm : REFERENCE TO DINT;
	p_diRevDlyTm : REFERENCE TO DINT;
	p_tMtrOffDlyTm : REFERENCE TO TIME;
	p_diTxInTimeOut : REFERENCE TO DINT;
	p_diTxOutTimeOut : REFERENCE TO DINT;
	p_eDirection : REFERENCE TO eConvDir;
	p_bGdBrdInit : REFERENCE TO BOOL;
	p_bGdBrdEnt : REFERENCE TO BOOL;
	p_sProgNm : REFERENCE TO STRING[15];
	p_tPshrExtTO : REFERENCE TO TIME;
	p_tPshrRetTO : REFERENCE TO TIME;
	p_tPullerExtTO : REFERENCE TO TIME;
	p_tPullerRetTO : REFERENCE TO TIME;
	p_tRotHomeTO : REFERENCE TO TIME;
	p_tRotRemoteTO : REFERENCE TO TIME;
	p_tRejectUpTO : REFERENCE TO TIME;
	p_tRejectDownTO : REFERENCE TO TIME;
	p_bNtSettingsLoadDone : REFERENCE TO BOOL;
END_VAR
(**)
(*Input*)
VAR
	p_bLeftSen : REFERENCE TO BOOL;
	p_bRightSen : REFERENCE TO BOOL;
	p_bMiddleSen : REFERENCE TO BOOL;
	p_bPullerChkSen : REFERENCE TO BOOL;
	p_bPshrExtSen : REFERENCE TO BOOL;
	p_bPshrRetSen : REFERENCE TO BOOL;
	p_bPshrExtSafetySen : REFERENCE TO BOOL;
	p_bPshrRetSafetySen : REFERENCE TO BOOL;
	p_bPullerExtSen : REFERENCE TO BOOL;
	p_bPullerRetSen : REFERENCE TO BOOL;
	p_bPullerExtSafetySen : REFERENCE TO BOOL;
	p_bPullerRetSafetySen : REFERENCE TO BOOL;
	p_bRotHomeSen : REFERENCE TO BOOL;
	p_bRotRemoteSen : REFERENCE TO BOOL;
	p_bRotHomeSafetySen : REFERENCE TO BOOL;
	p_bRotRemoteSafetySen : REFERENCE TO BOOL;
	p_bRejectUpSen : REFERENCE TO BOOL;
	p_bRejectDownSen : REFERENCE TO BOOL;
	p_bRejectUpSafetySen : REFERENCE TO BOOL;
	p_bRejectDownSafetySen : REFERENCE TO BOOL;
	p_bSelfTest : REFERENCE TO BOOL;
END_VAR
(*AutoRcp*)
VAR
	p_bNtParamAutoRcpPrep : REFERENCE TO BOOL;
	p_bMcParamAutoRcpDis : REFERENCE TO BOOL;
	p_eNtParamAutoRcpPrecededBy : REFERENCE TO eAutoRcpPreceded;
END_VAR
```

#### InputRef_Link.var
```iecst
(*2019-04-09*)
(**)
(*External Data*)
VAR
	p_bLinkOpsRun : REFERENCE TO BOOL;
END_VAR
(**)
VAR
	p_bLinkUIBypsInitConv : REFERENCE TO BOOL;
	p_bLinkDISafetyRlySig : REFERENCE TO BOOL;
	p_bLinkDIRgtSen : REFERENCE TO BOOL;
	p_bLinkDIClrSen : REFERENCE TO BOOL;
	p_usiLinkMcParamProdSelMcMod : REFERENCE TO USINT;
	p_eLinkOpsTravLifPosGo : REFERENCE TO eTravLifULPos;
	p_eLinkMcParamUSCommAMod : REFERENCE TO eMcSetCommMod;
	p_eLinkMcParamUSCommBMod : REFERENCE TO eMcSetCommMod;
	p_bLinkPshrRetSen : REFERENCE TO BOOL;
	p_bLinkPshrRetSlwSen : REFERENCE TO BOOL;
END_VAR
```

#### Local.var
```iecst
(*2019-06-17*)
VAR
	tylocalPshrConv : tyPshrConv;
END_VAR
(**)
(*Local Action, State & Status*)
VAR
	udiStatus : UDINT := 0;
	a_sStatText : ARRAY[0..60] OF STRING[200] := ['Idling','Initializing','Initializing With Reverse','Initializing With Pusher','Initializing With Puller','Initializing With Reject','Initializing With Inspection','Entering Board','Entering Board Until Inlet Signal Off','Entering Board With Reverse','Reversing Board','Reversing Board With Immediate Start Conv','Entering Board With Puller','Entering Board With Reject','Entering Board With Inspection','Pre Exiting Board','Resuming Reject Board',2('Exiting Board'),2('Exiting Board With Pusher'),'Pusher Setting All Control','Pusher Resetting All Control','Pusher Setting Extend','Pusher Setting Retract','Pusher Extending','Pusher Retracting','Puller Setting All Control','Puller Resetting All Control','Puller Setting Extend','Puller Setting Retract','Puller Extending','Puller Retracting','Rotating Setting All Control','Rotating Resetting All Control','Rotating Setting Home','Rotating Setting Remote','Rotating Turning Home','Rotating Turning Remote','Reject Setting All Control','Reject Resetting All Control','Reject Setting Up','Reject Setting Down','Reject Going Up','Reject Going Down','Stopping','Stopping With Pusher','Stopping With Puller','Stopping With Reject','Turning On Motor Signal','Turning On Motor Direction','Turning Off Motor Signal','Turning Off Motor Direction','Turning On All Motor Output','Turning Off All Motor Output',6('')];
END_VAR
(**)
(*Local Alarm*)
VAR
	tyAlmData : tyAlmDat;
END_VAR
(**)
(**)
(*Local*)
VAR
	bRstErr : BOOL;
	udiRstErrOld : UDINT;
	bInitDone : BOOL;
	bInitialDone : BOOL;
	usiStep : USINT;
	bInletOff : BOOL;
	fbWaitTm : TON := (PT:=T#1s);
	fbBoardOffTm : TON := (PT:=T#2s);
	eStatOld : eConvAction := ConvActIdle;
	fbInit : fbConvSenToSenTm;
	fbEnt : fbConvSenToSen;
	fbRev : fbConvSenToSenTm1;
	fbPreExit : fbConvSenToSenTm;
	fbExit : fbConvSenToSenOff;
	fbExit1 : fbConvSenToSenOff1;
	fbLongBrd : fbConvLongBrd;
	fbStop : fbConvMtrOff;
	fbPshrExtChk : fbPneuExtRetSenExtChk;
	fbPshrRetChk : fbPneuExtRetSenRetChk;
	fbPullerExtChk : fbPneuExtRetSenExtChk;
	fbPullerRetChk : fbPneuExtRetSenRetChk;
	fbRotHomeChk : fbPneuExtRetSenExtChk;
	fbRotRemoteChk : fbPneuExtRetSenRetChk;
	fbRejectUpChk : fbPneuExtRetSenExtChk;
	fbRejectDownChk : fbPneuExtRetSenRetChk;
	fbRightSenTm : TON := (PT:=T#1s);
	udiModuleNum : UDINT := 1501;
END_VAR
```

#### Act_Alarm.st
```iecst
(** 2019-03-25 **)
ACTION Act_Alarm:
	//Reset Error
	IF (tylocalPshrConv.Out.eStatus = Error) AND bRstErr THEN
		tylocalPshrConv.In.eAct	:= MagConv2ClpActIdle;
		tylocalPshrConv.Out.eStat	:= MagConv2ClpActIdle;
	END_IF

	IF tylocalPshrConv.In.udiRstErr <> udiRstErrOld THEN
		bRstErr			:= TRUE;
		udiRstErrOld	:= tylocalPshrConv.In.udiRstErr;
	ELSE
		bRstErr			:= FALSE;
	END_IF
	//Error
	IF EDGEPOS(tylocalPshrConv.Out.eStatus = Error) THEN

		tylocalPshrConv.Out.tyAlmData.udiCode		:= udiStatus;
		tylocalPshrConv.Out.tyAlmData.eSeverity		:= AlmSeverityError;
		tylocalPshrConv.Out.tyAlmData.udiRunTime	:= tylocalPshrConv.Out.tyAlmData.udiRunTime + 1;
		tylocalPshrConv.Out.tyAlmData.bAlm			:= TRUE;
		tylocalPshrConv.Out.tyAlmData.udiModuleNum  := udiModuleNum;
		g_sConvProgNm		    := tylocalUSSOT.In.sProgNm;

		tylocalPshrConv.Out.sStatTxt	:= tylocalPshrConv.Out.tyAlmData.sAlmMsg;

	ELSIF bRstErr AND (tyAlmData.udiCode <> 0) THEN

		tylocalPshrConv.Out.tyAlmData.udiCode	:= 0;
		tylocalPshrConv.Out.tyAlmData.eSeverity	:= AlmSeverityNA;
		tylocalPshrConv.Out.tyAlmData.bAlm			:= FALSE;
		tylocalPshrConv.Out.sStatTxt	:= a_sStatText[tylocalPshrConv.Out.eStat];

	END_IF

END_ACTION
```

#### Act_Background.st
```iecst
(** 2019-01-18 **)
ACTION Act_Background:

	IF p_bPshrExtSen = FALSE THEN
		bPshrExtended	:= FALSE;
	END_IF

	IF p_bPshrRetSen = FALSE THEN
		bPshrRetracted	:= FALSE;
	END_IF

	IF p_bPullerExtSen = FALSE THEN
		bPullerExtended	:= FALSE;
	END_IF

	IF p_bPullerRetSen = FALSE THEN
		bPullerRetracted	:= FALSE;
	END_IF

	IF p_bRotHomeSen = FALSE THEN
		bRotAtHome	:= FALSE;
	END_IF

	IF p_bRotRemoteSen = FALSE THEN
		bRotAtRemote	:= FALSE;
	END_IF

	IF p_bRejectUpSen = FALSE THEN
		bRejectAtUp	:= FALSE;
	END_IF

	IF p_bRejectDownSen = FALSE THEN
		bRejectAtDown	:= FALSE;
	END_IF

	//ADDED
	IF p_eAct <> ConvActExitPshr  THEN
		bPshrRetAllwTraverse :=   FALSE;
	ELSIF bPshrRetCtrl AND p_bLinkPshrRetSlwSen THEN
		bPshrRetAllwTraverse :=   TRUE;
	END_IF

END_ACTION
```

#### Act_InitGlobal.st
```iecst
(** 2019-04-09 **)
ACTION Act_InitGlobal:

	(* Always Change If Project Change *)

	//Pass Data To Link
	p_bLinkOpsRun ACCESS p_OpsRun;

	p_bLinkUIBypsInitConv ACCESS p_UIOpsBypsInitConv;
	p_bLinkDISafetyRlySig ACCESS p_DISafetyRlySig;
	p_bLinkDIRgtSen ACCESS p_DIConvRgtSen;
	p_bLinkDIClrSen ACCESS p_DIConvClrSen;
//	p_usiLinkMcParamProdSelMcMod ACCESS p_ProdRcpCurrRcp1McMod;
	p_eLinkOpsTravLifPosGo ACCESS p_OpsTravLifULPosGo;
	p_eLinkMcParamUSCommAMod ACCESS p_McParamUSCommAMod;
	p_eLinkMcParamUSCommBMod ACCESS p_McParamUSCommBMod;
	p_bLinkPshrRetSen ACCESS p_DIPusherRetRS;
	p_bLinkPshrRetSlwSen ACCESS p_DIPusherRetSlwSen;

	//Pass Data To Internal Use
	p_udiRstErr ACCESS p_RstErrReset;
	p_bManual ACCESS p_UIMnlMod;
	p_bOnDirMod ACCESS p_NtParamPshrConvOnDirMod;
	p_diInitTm ACCESS p_McParamConvInitTm;
	p_tMtrOffDlyTm ACCESS p_NtParamPshrConvMtrOffDlyTm;
	p_diTxInTimeOut ACCESS p_McParamTranInErrDlyTm;
	p_eDirection ACCESS p_NtParamProjConvDir;
	p_sProgNm ACCESS p_NtParamPshrConvProgNm;
	p_tPshrExtTO ACCESS p_NtParamPshrConvPshrExtTO;
	p_tPshrRetTO ACCESS p_NtParamPshrConvPshrRetTO;
	p_bLeftSen ACCESS p_DIConvLftSen;
	p_bMiddleSen ACCESS p_DIConvMidSen;
	p_bPshrExtSen ACCESS p_DIPusherExtRS;
//	p_bPshrRetSen ACCESS p_DIPusherRetSlwSen;
	p_bNtSettingsLoadDone ACCESS p_StartupNtSettingsLoadDone;

	p_bSelfTest ACCESS p_OpsTravLifULSelfTest;

	p_bNtParamAutoRcpPrep ACCESS p_NtParamAutoRcpPrep;
	p_bMcParamAutoRcpDis  ACCESS p_McParamAutoRcpDisable;
	p_eNtParamAutoRcpPrecededBy ACCESS p_NtParamAutoRcpPrecededBy;
	(* Always Change If Project Change *)

END_ACTION
```

#### Act_Initial.st
```iecst
(** 2019-03-22 **)
ACTION Act_Initial:

	//Initial
	tylocalPshrConv.Out.sStatTxt	:= a_sStatText[eStat];

	fbWaitTm(IN := FALSE);

	fbInit.bStartSen	:= TRUE;
	fbInit(bEn := FALSE);

	fbEnt.bStartSen		:= TRUE;
	fbEnt(bEn := FALSE);

	fbRev(bEn := FALSE);

	fbPreExit.bStartSen		:= TRUE;
	fbPreExit(bEn := FALSE);

	fbExit.bStartSen	:= TRUE;
	fbExit(bEn := FALSE);

	fbExit1.bStartSen		:= TRUE;
	fbExit1(bEn := FALSE);

	fbStop(bEn := FALSE);

	fbPshrExtChk(bEn := FALSE);

	fbPshrRetChk(bEn := FALSE);

	fbPullerExtChk(bEn := FALSE);

	fbPullerRetChk(bEn := FALSE);

	fbRotHomeChk(bEn := FALSE);

	fbRotRemoteChk(bEn := FALSE);

	fbRejectUpChk(bEn := FALSE);

	fbRejectDownChk(bEn := FALSE);

END_ACTION
```

#### Act_InputConfig.st
```iecst
(** 2019-04-09 **)
ACTION Act_InputConfig:

	(* Always Change If Project Change *)

	//Pass Data To Link

	tylocalPshrConv.In.bLinkUIBypsInitConv := g_tyUIOpsByps.bInitConv;
	tylocalPshrConv.In.bLinkDISafetyRlySig := g_tyDInput.bSafetyRlySig;
	tylocalPshrConv.In.bLinkDIRgtSen := g_tyDInput.bConvRgtSen;
	tylocalPshrConv.In.bLinkDIClrSen := g_tyDInput.bConvClrSen;
//	tylocalPshrConv.In.usiLinkMcParamProdSelMcMod := g_tyProdRcpCurrRcp1McMod;
	tylocalPshrConv.In.eLinkOpsTravLifPosGo := g_tyOpsTravLifUL.eTravLifPosGo;
	tylocalPshrConv.In.eLinkMcParamUSCommAMod := g_tyMcParamCurr.eUSCommAMod;
	tylocalPshrConv.In.eLinkMcParamUSCommBMod := g_tyMcParamCurr.eUSCommBMod;
	tylocalPshrConv.In.bLinkPshrRetSen := g_tyDInput.bPusherRetRS;
	tylocalPshrConv.In.bLinkPshrRetSlwSen := g_tyDInput.bPusherRetSlwSen;

	//Pass Data To Internal Use
	tylocalPshrConv.In.udiRstErr := g_tyRstErr.bReset;
	tylocalPshrConv.In.bManual := g_tyUIOut.bManualMod;
	tylocalPshrConv.In.bOnDirMod := g_tyNtParamCurr.bPshrConvOnDirMod;
	tylocalPshrConv.In.diInitTm := g_tyMcParamCurr.tConvInitTm;
	tylocalPshrConv.In.tMtrOffDlyTm := g_tyNtParamCurr.tPshrConvMtrOffDlyTm;
	tylocalPshrConv.In.diTxInTimeOut := g_tyMcParamCurr.tTranInErrDlyTm;
	tylocalPshrConv.In.eDirection := g_tyNtParamCurr.bProjConvDir;
	tylocalPshrConv.In.sProgNm := g_tyNtParamCurr.sPshrConvProgNm;
	tylocalPshrConv.In.tPshrExtTO := g_tyNtParamCurr.tPshrConvPshrExtTO;
	tylocalPshrConv.In.tPshrRetTO := g_tyNtParamCurr.tPshrConvPshrRetTO;
	tylocalPshrConv.In.bLeftSen := g_tyDInput.bConvLftSen;
	tylocalPshrConv.In.bMiddleSen := g_tyDInput.bConvMidSen;
	tylocalPshrConv.In.bPshrExtSen := g_tyDInput.bPusherExtRS;
//	tylocalPshrConv.In.bPshrRetSen := g_tyDInput.bPusherRetSlwSen;

	tylocalPshrConv.In.bSelfTest := g_tyOpsTravLifUL.bSelfTest;

	tylocalPshrConv.In.bNtParamAutoRcpPrep := g_tyNtParamCurr.bAutoRcpPrep;
	tylocalPshrConv.In.bMcParamAutoRcpDis  := g_tyMcParamCurr.bAutoRcpDisable;
	(* Always Change If Project Change *)

	IF g_tyOps.bRun = TRUE THEN
		tylocalPshrConv.In.eAct := g_tyOpsTravLifUL.eConvAct;
	ELSIF tylocalPshrConv.In.bManual = TRUE THEN
		tylocalPshrConv.In.eAct := g_tyUIOut.eMnlAct.ePshrConvAct;
	ELSE
		tylocalPshrConv.In.eAct := eAct;
	END_IF
END_ACTION
```

#### Act_Link.st
```iecst
(** 2019-03-29 **)
ACTION Act_Link:

	IF tylocalPshrConv.In.bNtParamAutoRcpPrep AND NOT(tylocalPshrConv.In.bMcParamAutoRcpDis) THEN //AutoRcp Ignored Follower
		tylocalPshrConv.In.usiLinkMcParamProdSelMcMod ACCESS tylocalPshrConv.In.ProdRcpCurrRcp0McMod;
	ELSE
		tylocalPshrConv.In.usiLinkMcParamProdSelMcMod ACCESS tylocalPshrConv.In.ProdRcpCurrRcp1McMod;
	END_IF

	IF tylocalPshrConv.In.bLinkDISafetyRlySig = FALSE OR tylocalPshrConv.Out.eStatus = Error  THEN
		tylocalPshrConv.Out.bPshrExtCtrl		:= FALSE;
		tylocalPshrConv.Out.bPshrRetCtrl		:= FALSE;
		tylocalPshrConv.Out.bPshrExtended		:= FALSE;
		tylocalPshrConv.Out.bPshrRetracted		:= FALSE;

		tylocalPshrConv.Out.bPullerExtCtrl		:= FALSE;
		tylocalPshrConv.Out.bPullerRetCtrl		:= FALSE;
		tylocalPshrConv.Out.bPullerExtended		:= FALSE;
		tylocalPshrConv.Out.bPullerRetracted	:= FALSE;

		tylocalPshrConv.Out.bRotRemoteCtrl		:= FALSE;
		tylocalPshrConv.Out.bRotAtRemote		:= FALSE;
		tylocalPshrConv.Out.bRotAtHome			:= FALSE;

		tylocalPshrConv.Out.bRejectUpCtrl		:= FALSE;
		tylocalPshrConv.Out.bRejectDownCtrl		:= FALSE;
		tylocalPshrConv.Out.bRejectAtUp			:= FALSE;
		tylocalPshrConv.Out.bRejectAtDown		:= FALSE;
	END_IF

	//Bypass Intializing Conveyor
	IF tylocalPshrConv.In.bLinkUIBypsInitConv THEN
		tylocalPshrConv.In.diInitTm ACCESS ADR(diInitTm);
	ELSE
		tylocalPshrConv.In.diInitTm ACCESS tylocalPshrConv.In.McParamConvInitTm;
	END_IF

	fbRightSenTm(IN:= tylocalPshrConv.Out.bMtrSigOnOrLToR AND tylocalPshrConv.In.bRightSen = FALSE, PT:= DINT_TO_TIME(tylocalPshrConv.In.diInitTm - 1000));
	//Sensor
	IF tylocalPshrConv.In.bSelfTest = FALSE THEN
		tylocalPshrConv.In.bRightSen	:= tylocalPshrConv.In.bLinkDIRgtSen OR tylocalPshrConv.In.bLinkDIClrSen; //previously this part block for safety
		fbBoardOffTm(IN:= tylocalPshrConv.In.bLeftSen = FALSE AND tylocalPshrConv.In.bRightSen = FALSE AND tylocalPshrConv.Out.bMtrDirOrRToL = FALSE AND tylocalPshrConv.Out.bMtrSigOnOrLToR = FALSE);
		IF EDGEPOS(fbBoardOffTm.Q) THEN
			tylocalPshrConv.Out.bHvBrd := FALSE;
		END_IF
	ELSE
		IF fbRightSenTm.Q THEN
			tylocalPshrConv.In.bRightSen := TRUE;
		ELSIF tylocalPshrConv.In.bPshrExtSen THEN
			tylocalPshrConv.In.bRightSen := FALSE;
		END_IF
	END_IF

	tylocalPshrConv.In.bPshrRetSen := tylocalPshrConv.In.bLinkPshrRetSen; // OR tylocalPshrConv.In.bLinkPshrRetSlwSen;

	//Good Board Init
	CASE tylocalPshrConv.In.usiLinkMcParamProdSelMcMod OF
		ULModUnloadFrontLnA, ULModUnloadRearLnB, ULModUnloadDualLnAB:
			tylocalPshrConv.In.bGdBrdEnt	:= TRUE;
		ULModRejFrontLnA, ULModRejFrontLnARev, ULModRejRearLnB, ULModRejRearLnBRev, ULModRejDualLnA, ULModRejDualLnB:
			tylocalPshrConv.In.bGdBrdEnt	:= FALSE;
	END_CASE

	//Good Board Enter
	IF tylocalPshrConv.In.eLinkOpsTravLifPosGo = TravLifULPosUS1 THEN

		IF tylocalPshrConv.In.eLinkMcParamUSCommAMod = McSetCommModSMEMA THEN
			tylocalPshrConv.In.bGdBrdEnt := g_tyUSSMEMAA.bUSGdBrdRdy;
		ELSIF tylocalPshrConv.In.eLinkMcParamUSCommAMod = McSetCommModHermes THEN
			tylocalPshrConv.In.bGdBrdEnt := g_tyUSHermesA.bUSGdRdy;
		END_IF

	ELSIF tylocalPshrConv.In.eLinkOpsTravLifPosGo = TravLifULPosUS2 THEN

		IF tylocalPshrConv.In.eLinkMcParamUSCommBMod = McSetCommModSMEMA THEN
			tylocalPshrConv.In.bGdBrdEnt := g_tyUSSMEMAB.bUSGdBrdRdy;
		ELSIF tylocalPshrConv.In.eLinkMcParamUSCommBMod = McSetCommModHermes THEN
			tylocalPshrConv.In.bGdBrdEnt := g_tyUSHermesB.bUSGdRdy;
		END_IF

	END_IF

END_ACTION
```

#### Act_LinkAction.st
```iecst
(** 2019-04-09 **)
ACTION Act_LinkAction:

	IF p_bLinkOpsRun = TRUE THEN
		p_eAct ACCESS p_OpsTravLifULConvAct;
	ELSIF p_bManual = TRUE THEN
		p_eAct ACCESS p_UIPshrConvAct;
	ELSE
		p_eAct ACCESS ADR(eAct);
	END_IF

END_ACTION
```
